// TIA Portal project "SWNC V1.0 pulldown" (V16)

(* hardware
DEVICE "S7-1200 station_1"  S7-1200 Station
   slot 0: "Rack_0"  S7-1200 Rack  Rack  V1.0
   slot 1: "PLC_1"  CPU 1214C DC/DC/DC  6ES7 214-1AG40-0XB0  V4.4
   slot 2: "DI 8x24VDC_1"  6ES7 221-1BF32-0XB0  V2.0
   slot 3: "CB 1241 (RS485)"  CB 1241 (RS485)  6ES7 241-1CH30-1XB0  V1.0
   slot 3: "DQ 8xRelay_1"  SM 1222 DQ8 x relay  6ES7 222-1HF32-0XB0  V2.0
   slot 4: "AI 8x13BIT_1"  6ES7 231-4HF32-0XB0  V2.1
   slot 5: "AQ 2x14BIT_1"  SM 1232 AQ2  6ES7 232-4HB32-0XB0  V2.1
DEVICE "HMI_1"  KTP700 Basic PN
   slot 0: "HMI_1"  KTP700 Basic PN  6AV2 123-2GB03-0AX0  16.0.0.0
   slot 1: "HMI_RT_1"  KTP700 Basic PN  6AV2 123-2GB03-0AX0  16.0.0.0
   slot 5: "HMI_1.IE_CP_1"  PROFINET Interface  16.0.0.0
      slot 1: "PROFINET Interface_1"  PROFINET Interface
         slot 1: "Port_1"  Port
*)

// ===== PLC "PLC_1"  CPU 1214C DC/DC/DC =====

VAR_GLOBAL   // PLC tag table "Default tag table"
   "HOA Manual" AT %I0.5 : Bool;
   "HOA Auto Run" AT %I0.4 : Bool;
   "supply empty" AT %I0.7 : Bool;
   "chiller full" AT %I1.0 : Bool;
   "chiller empty" AT %I1.1 : Bool;
   "inside full" AT %I1.3 : Bool;
   "inside discharge" AT %I1.4 : Bool;
   "inside empty" AT %I1.5 : Bool;
   "outside full" AT %I2.0 : Bool;
   "outside discharge" AT %I2.1 : Bool;
   "outside empty" AT %I2.2 : Bool;
   "purge full" AT %I1.2 : Bool;
   "E-Stop_Panel_pushed" AT %I0.6 : Bool;   // true when Estop is pushed
   "Run_button" AT %I0.0 : Bool;
   "Stop_reset_button" AT %I0.1 : Bool;
   "MAN 1 (Outside)" AT %Q0.0 : Bool;   // NO - to chiller NC - to purge
   "MAN 2 (Inside)" AT %Q0.1 : Bool;   // NO - to Purge NC - to Outside
   "MAN 3 (Supply)" AT %Q0.2 : Bool;   // NO - to outside NC - to inside
   "MAN 4 (Not Used)" AT %Q0.3 : Bool;   // NO - to outside NC - to inside
   "Pump 1 Outside cooling" AT %Q0.4 : Bool;
   "Pump 2 Outside Out" AT %Q0.5 : Bool;
   "Pump 3 Inside Cooling" AT %Q0.6 : Bool;
   "Pump 4 Inside Out" AT %Q0.7 : Bool;
   "Pump 5 Chiller out" AT %Q1.0 : Bool;
   "Pump 6 Supply out" AT %Q1.1 : Bool;
   "Pump 7 HX pump" AT %Q12.0 : Bool;
   "Pump 8 Purge out" AT %Q12.1 : Bool;
   "System_Byte" AT %MB1000 : Byte;
   "FirstScan" AT %M1000.0 : Bool;
   "DiagStatusUpdate" AT %M1000.1 : Bool;
   "AlwaysTRUE" AT %M1000.2 : Bool;
   "AlwaysFALSE" AT %M1000.3 : Bool;
   "Clock_Byte" AT %MB1001 : Byte;
   "Clock_10Hz" AT %M1001.0 : Bool;
   "Clock_5Hz" AT %M1001.1 : Bool;
   "Clock_2.5Hz" AT %M1001.2 : Bool;
   "Clock_2Hz" AT %M1001.3 : Bool;
   "Clock_1.25Hz" AT %M1001.4 : Bool;
   "Clock_1Hz" AT %M1001.5 : Bool;
   "Clock_0.625Hz" AT %M1001.6 : Bool;
   "Clock_0.5Hz" AT %M1001.7 : Bool;
   "Mode Bit" AT %MB0 : USInt;
   "HOA Off" AT %M1.0 : Bool;
   "Outside Fan" AT %M1.3 : Bool;
   "Inside Fan" AT %M1.4 : Bool;
   "Outside Cooling" AT %M1.5 : Bool;
   "Inside Cooling" AT %M1.6 : Bool;
   "pump out supply" AT %M1.7 : Bool;
   "pump out Chiller" AT %M2.0 : Bool;
   "pump out inside tank" AT %M2.1 : Bool;
   "Pump out outside tank" AT %M2.2 : Bool;
   "pump out purge tank" AT %M2.3 : Bool;
   "pump chiller circulation" AT %M2.4 : Bool;
   "valve from supply" AT %M2.5 : Bool;   // 0 = to outdoor 1= to indoor
   "valve from chiller" AT %M2.6 : Bool;   // 0 = to outdoor 1= to indoor
   "valve from inside" AT %M2.7 : Bool;   // 0 = to purge 1= to chiller
   "valve from outside" AT %M3.0 : Bool;   // 0 = to purge 1= to chiller
   "chiller enable" AT %M3.1 : Bool;
   "SB OUTSIDE COOLING" AT %M3.2 : Bool;
   "SB INSIDE COOLING" AT %M3.3 : Bool;
   "SB pump out supply" AT %M3.4 : Bool;
   "SB pump out Chiller" AT %M3.5 : Bool;
   "SB pump out inside tank" AT %M3.6 : Bool;
   "SB Pump out outside tank" AT %M3.7 : Bool;
   "SB pump out purge tank" AT %M4.0 : Bool;
   "SB pump chiller circulation" AT %M4.1 : Bool;
   "SB valve from supply" AT %M4.2 : Bool;
   "SB valve from chiller" AT %M4.3 : Bool;
   "SB valve from inside" AT %M4.4 : Bool;
   "SB valve from outside" AT %M4.5 : Bool;
   "SB chiller enable" AT %M4.6 : Bool;
   "SB INSIDE FAN" AT %M4.7 : Bool;
   "SB OUTSIDE FAN" AT %M5.0 : Bool;
   "inside change bit" AT %M5.1 : Bool;   // true when tank change is in progress
   "PB_chill to regen trans" AT %M5.2 : Bool;
   "PB_regen to chill trans" AT %M5.3 : Bool;
   "Emergency_flags" AT %MW6 : Int;   // Contain all the Estop scenarios. 1=active, 0=inactive
   "Emergency_check" AT %M7.0 : Bool;   // ON when any emergency scenario occurs
   "Emergency_Ack" AT %M1.2 : Bool;
   "Alarm_Ack" AT %MW1002 : Int;
   "global MB address" AT %MB8 : SInt;
   "GET_INT" AT %MW12 : Int;
   "HTS1" AT %M5.4 : Bool;   // Set bit for HT sensors
   "HTS3" AT %M5.6 : Bool;
   "HTS4" AT %M5.7 : Bool;
   "HTS2" AT %M9.0 : Bool;
   "DGS1" AT %M5.5 : Bool;   // Depth Gauge set bit
   "DGS2" AT %M9.1 : Bool;
   "WTSB" AT %M9.2 : Bool;   // Water temp set bit
   "THE TIME" AT %MD14 : Time_Of_Day;
   "Global GH Temp" AT %MD18 : Real;
   "Global GH Hum" AT %MD22 : Real;
   "Program Run" AT %M1.1 : Bool;
   "Regen bit" AT %M9.3 : Bool;
   "Auto time override" AT %M9.4 : Bool;
   "Manual day night toggle" AT %M9.5 : Bool;
   "Manual night to day trans" AT %M9.6 : Bool;
   "Manual day to night trans" AT %M9.7 : Bool;
   "time OS1" AT %M10.0 : Bool;
   "time OS2" AT %M10.1 : Bool;
   "time OS3" AT %M10.2 : Bool;
   "time OS4" AT %M10.3 : Bool;
   "WSSB" AT %M10.4 : Bool;
   "log start" AT %M10.5 : Bool;
   "log start lock" AT %M10.6 : Bool;
END_VAR

DATA_BLOCK "System Properties"   // DB1
{ S7_Optimized_Access := 'TRUE' }
VERSION : 0.1
   VAR
      "Time" : Struct
         "Current Time" : Time_Of_Day;
         "Night time start" : Time_Of_Day := TOD#20:00:00;
         "Night time end" : Time_Of_Day := TOD#06:00:00;
         "is it day???" : Bool;   // 1 = day, 0 = night
      END_STRUCT;
      "Situation Bits" : Struct
         HOA : Int;
         "Day Run" : Bool;
         "Night Run" : Bool;
         "Day Tank Change" : Int;
         "Night Regen Complete" : Bool;
         "Day/Night Transition Bit" : Int;   // 0= no trans 1= day to night 2= night to day
         "regen or chill" : Int;   // 0 = chill , 1 = regen 3 = transition in progress
         "chilling to regen transition" : Bool;
         "regen to chilling transition" : Bool;
      END_STRUCT;
      "Comment status" : String := 'Idle';
      "Comment DN" : String := 'Time Unknown';
   END_VAR
BEGIN
END_DATA_BLOCK

DATA_BLOCK "Outputs"   // DB2
{ S7_Optimized_Access := 'TRUE' }
VERSION : 0.1
   VAR
      Fans : Struct
         "Inside Fan" : Bool;
         "Outside Fan" : Bool;
      END_STRUCT;
      "Cooling Pad Pumps" : Struct
         "Inside Cooling" : Bool;
         "Outside Cooling" : Bool;
      END_STRUCT;
      Pumps : Struct
         "From Supply Tank" : Bool;
         "From Chiller Tank" : Bool;
         "From Inside Tank" : Bool;
         "From Outside Tank" : Bool;
         "From Purge Tank" : Bool;
         "Chiller Recirculation" : Bool;
      END_STRUCT;
      Valves : Struct
         "From Supply" : Bool;   // 0= to outdoor, 1= to indoor
         "From Chiller" : Bool;   // 0= to outdoor, 1= to indoor
         "From Indoor" : Bool;   // 0= to Purge, 1= to Chiller
         "From Outdoor" : Bool;   // 0= to Purge, 1= to Chiller
      END_STRUCT;
      Chiller : Struct
         "Chiller Enable" : Bool;
      END_STRUCT;
   END_VAR
BEGIN
END_DATA_BLOCK

DATA_BLOCK "Alarm Conditions"   // DB3
{ S7_Optimized_Access := 'TRUE' }
VERSION : 0.1
   VAR
      "E Stop Pushed" : Bool;
      "Pump Over run" : Bool;
      "Alarm bit" : Bool;
      "Alarm Reset" : Bool;
   END_VAR
BEGIN
END_DATA_BLOCK

DATA_BLOCK "What Time is it?_DB"   // DB4
{ S7_Optimized_Access := 'TRUE' }
VERSION : 0.1
// stored: InstanceOfName What Time is it?
"What Time is it?"
BEGIN
END_DATA_BLOCK

DATA_BLOCK "What mode_DB"   // DB5
{ S7_Optimized_Access := 'TRUE' }
VERSION : 0.1
// stored: InstanceOfName What mode
"What mode"
BEGIN
END_DATA_BLOCK

DATA_BLOCK "Manual Mode_DB"   // DB6
{ S7_Optimized_Access := 'TRUE' }
VERSION : 0.1
// stored: InstanceOfName Manual Mode
"Manual Mode"
BEGIN
END_DATA_BLOCK

DATA_BLOCK "Day Operation_DB"   // DB7
{ S7_Optimized_Access := 'TRUE' }
VERSION : 0.1
// stored: InstanceOfName Day Operation
"Day Operation"
BEGIN
END_DATA_BLOCK

DATA_BLOCK "Night Operation_DB"   // DB8
{ S7_Optimized_Access := 'TRUE' }
VERSION : 0.1
// stored: InstanceOfName Night Operation
"Night Operation"
BEGIN
END_DATA_BLOCK

DATA_BLOCK "Tank check_DB"   // DB9
{ S7_Optimized_Access := 'TRUE' }
VERSION : 0.1
// stored: InstanceOfName Tank check
"Tank check"
BEGIN
END_DATA_BLOCK

DATA_BLOCK "inside tank switch_DB"   // DB11
{ S7_Optimized_Access := 'TRUE' }
VERSION : 0.1
// stored: InstanceOfName inside tank switch
"inside tank switch"
BEGIN
END_DATA_BLOCK

DATA_BLOCK "Auto Run Program_DB"   // DB12
{ S7_Optimized_Access := 'TRUE' }
VERSION : 0.1
// stored: InstanceOfName Auto Run Program
"Auto Run Program"
BEGIN
END_DATA_BLOCK

DATA_BLOCK "Day to Night change_DB"   // DB13
{ S7_Optimized_Access := 'TRUE' }
VERSION : 0.1
// stored: InstanceOfName Day to Night change
"Day to Night change"
BEGIN
END_DATA_BLOCK

DATA_BLOCK "Night to Day change_DB"   // DB14
{ S7_Optimized_Access := 'TRUE' }
VERSION : 0.1
// stored: InstanceOfName Night to Day change
"Night to Day change"
BEGIN
END_DATA_BLOCK

DATA_BLOCK "Auto Time_DB"   // DB15
{ S7_Optimized_Access := 'TRUE' }
VERSION : 0.1
// stored: InstanceOfName Auto Time
"Auto Time"
BEGIN
END_DATA_BLOCK

DATA_BLOCK "Manual Time_DB"   // DB18
{ S7_Optimized_Access := 'TRUE' }
VERSION : 0.1
// stored: InstanceOfName Manual Time
"Manual Time"
BEGIN
END_DATA_BLOCK

DATA_BLOCK "Get Weather Station Data_DB"   // DB20
{ S7_Optimized_Access := 'TRUE' }
VERSION : 0.1
// stored: InstanceOfName Get Weather Station Data
"Get Weather Station Data"
BEGIN
END_DATA_BLOCK

DATA_BLOCK "Weather Station Data"   // DB21
{ S7_Optimized_Access := 'TRUE' }
VERSION : 0.1
   VAR
      "Air Temperature" : Real;
      "Air Humidity" : Real;
      "Air Pressure (mBar)" : Real;
      CO2 : Real;
      "PM 2.5" : Real;
      "PM 10" : Real;
      "PM 100" : Real;
      "Wind Speed" : Real;
      "Wind Direction" : Real;
      "Light Intensity (μmol/m^2.s)" : Real;
      "Current Rainfall" : Real;
   END_VAR
BEGIN
END_DATA_BLOCK

DATA_BLOCK "Emergency_Stop_DB"   // DB22
{ S7_Optimized_Access := 'TRUE' }
AUTHOR : FF
VERSION : 0.1
// stored: InstanceOfName Emergency_Stop
"Emergency_Stop"
BEGIN
END_DATA_BLOCK

DATA_BLOCK "MODBUS DATA"   // DB24
{ S7_Optimized_Access := 'FALSE' }
VERSION : 0.1
   VAR
      "Start up done" : Bool;
      "Master Busy" : Bool;
      "Master Done" : Bool;
      "Master Error" : Bool;
      "Slave Address" : Int;
      "Memory Address" : DInt;
      "read/write" : Int;
      "data length" : Int;
      "memory pointer" : Byte;
   END_VAR
BEGIN
END_DATA_BLOCK

DATA_BLOCK "Ts and Hs"   // DB26
{ S7_Optimized_Access := 'TRUE' }
VERSION : 0.1
   VAR
      "Ambient Temp" : Real;
      "Ambient Humidity" : Real;
      "GH Temp" : Real;
      "GH Humidity" : Real;
      "Outside Outlet Temp" : Real;
      "Outside Outlet  Humidity" : Real;
      "Inside Outlet Temp" : Real;
      "Inside Outlet Humidity" : Real;
      "Chiller Tank Water Temp" : Real;
   END_VAR
BEGIN
END_DATA_BLOCK

DATA_BLOCK "MODBUS REGISTER"   // DB27
{ S7_Optimized_Access := 'FALSE' }
VERSION : 0.1
   VAR
      "Incomiong/Outgoing data" : Array[0..20] of Int;
   END_VAR
BEGIN
END_DATA_BLOCK

DATA_BLOCK "MODBUS_DB"   // DB28
{ S7_Optimized_Access := 'TRUE' }
VERSION : 0.1
// stored: InstanceOfName MODBUS
"MODBUS"
BEGIN
END_DATA_BLOCK

DATA_BLOCK "Get Ts and Hs_DB"   // DB29
{ S7_Optimized_Access := 'TRUE' }
VERSION : 0.1
// stored: InstanceOfName Get Ts and Hs
"Get Ts and Hs"
BEGIN
END_DATA_BLOCK

DATA_BLOCK "Depth Readings"   // DB30
{ S7_Optimized_Access := 'TRUE' }
VERSION : 0.1
   VAR
      "Outside Tank Depth" : Real;
      "Inside Tank Depth" : Real;
   END_VAR
BEGIN
END_DATA_BLOCK

DATA_BLOCK "Get Depths_DB"   // DB32
{ S7_Optimized_Access := 'TRUE' }
VERSION : 0.1
// stored: InstanceOfName Get Depths
"Get Depths"
BEGIN
END_DATA_BLOCK

DATA_BLOCK "Get Water Temp_DB"   // DB33
{ S7_Optimized_Access := 'TRUE' }
VERSION : 0.1
// stored: InstanceOfName Get Water Temp
"Get Water Temp"
BEGIN
END_DATA_BLOCK

DATA_BLOCK "Setup"   // DB34
{ S7_Optimized_Access := 'TRUE' }
VERSION : 0.1
   VAR
      "Day Cooling on/off threshold" : Real := 20.0;
      "Night Cooling on/off threshold" : Real := 18.0;
      "Regen hum low" : Real := 35.0;
      "Regen hum high" : Real := 65.0;
      "Day Fan Speed" : Int := 6000;
      "Night Fan Speed" : Int := 1000;
   END_VAR
BEGIN
END_DATA_BLOCK

DATA_BLOCK "Update Outside Fan_DB"   // DB35
{ S7_Optimized_Access := 'TRUE' }
VERSION : 0.1
// stored: InstanceOfName Update Outside Fan
"Update Outside Fan"
BEGIN
END_DATA_BLOCK

DATA_BLOCK "Update Inside Fan_DB"   // DB36
{ S7_Optimized_Access := 'TRUE' }
VERSION : 0.1
// stored: InstanceOfName Update Inside Fan
"Update Inside Fan"
BEGIN
END_DATA_BLOCK

DATA_BLOCK "MODBUS_DB_1"   // DB37
{ S7_Optimized_Access := 'TRUE' }
VERSION : 0.1
// stored: InstanceOfName MODBUS
"MODBUS"
BEGIN
END_DATA_BLOCK

DATA_BLOCK "Inside Fan Emergancy_DB"   // DB38
{ S7_Optimized_Access := 'TRUE' }
VERSION : 0.1
// stored: InstanceOfName Inside Fan Emergancy
"Inside Fan Emergancy"
BEGIN
END_DATA_BLOCK

DATA_BLOCK "MODBUS_DB_2"   // DB39
{ S7_Optimized_Access := 'TRUE' }
VERSION : 0.1
// stored: InstanceOfName MODBUS
"MODBUS"
BEGIN
END_DATA_BLOCK

DATA_BLOCK "MODBUS_DB_3"   // DB40
{ S7_Optimized_Access := 'TRUE' }
VERSION : 0.1
// stored: InstanceOfName MODBUS
"MODBUS"
BEGIN
END_DATA_BLOCK

DATA_BLOCK "Outside Fan Emergancy_DB"   // DB41
{ S7_Optimized_Access := 'TRUE' }
VERSION : 0.1
// stored: InstanceOfName Outside Fan Emergancy
"Outside Fan Emergancy"
BEGIN
END_DATA_BLOCK

DATA_BLOCK "Update Outside Fan_DB_1"   // DB42
{ S7_Optimized_Access := 'TRUE' }
VERSION : 0.1
// stored: InstanceOfName Update Outside Fan
"Update Outside Fan"
BEGIN
END_DATA_BLOCK

DATA_BLOCK "MODBUS_DB_4"   // DB43
{ S7_Optimized_Access := 'TRUE' }
VERSION : 0.1
// stored: InstanceOfName MODBUS
"MODBUS"
BEGIN
END_DATA_BLOCK

DATA_BLOCK "Off Mode_DB"   // DB44
{ S7_Optimized_Access := 'TRUE' }
VERSION : 0.1
// stored: InstanceOfName Off Mode
"Off Mode"
BEGIN
END_DATA_BLOCK

DATA_BLOCK "Fan Speeds"   // DB48
{ S7_Optimized_Access := 'TRUE' }
VERSION : 0.1
   VAR
      "Inside Fan Speed" : Int := 6000;
      "Outside Fan Speed" : Int := 6000;
   END_VAR
BEGIN
END_DATA_BLOCK

DATA_BLOCK "Current States"   // DB49
{ S7_Optimized_Access := 'TRUE' }
VERSION : 0.1
BEGIN
END_DATA_BLOCK

DATA_BLOCK "From AWS"   // DB50
{ S7_Optimized_Access := 'TRUE' }
VERSION : 0.1
BEGIN
END_DATA_BLOCK

DATA_BLOCK "Data log setup"   // DB52
{ S7_Optimized_Access := 'TRUE' }
VERSION : 0.1
   VAR
      "name" : String := 'Ashs_Log_Overnight';
      ID : DInt;
      hedder : String := 'Out Temp,Out Hum,In Temp,In Hum';
      "data log data" : Struct
         data : Array[0..3] of Real;
      END_STRUCT;
      "start done" : Bool;
   END_VAR
BEGIN
END_DATA_BLOCK

DATA_BLOCK "Data logging main_DB"   // DB54
{ S7_Optimized_Access := 'TRUE' }
VERSION : 0.1
// stored: InstanceOfName Data logging main
"Data logging main"
BEGIN
END_DATA_BLOCK

// folder: System blocks/Program resources

DATA_BLOCK "IEC_Timer_0_DB"   // DB10
{ S7_Optimized_Access := 'TRUE' }
AUTHOR : Simatic
FAMILY : IEC
NAME : IEC_TMR
VERSION : 1.0
// stored: InstanceOfName IEC_TIMER
"IEC_TIMER"
BEGIN
END_DATA_BLOCK

DATA_BLOCK "IEC_Timer_0_DB_2"   // DB16
{ S7_Optimized_Access := 'TRUE' }
AUTHOR : Simatic
FAMILY : IEC
NAME : IEC_TMR
VERSION : 1.0
// stored: InstanceOfName IEC_TIMER
"IEC_TIMER"
BEGIN
END_DATA_BLOCK

DATA_BLOCK "IEC_Timer_0_DB_3"   // DB17
{ S7_Optimized_Access := 'TRUE' }
AUTHOR : Simatic
FAMILY : IEC
NAME : IEC_TMR
VERSION : 1.0
// stored: InstanceOfName IEC_TIMER
"IEC_TIMER"
BEGIN
END_DATA_BLOCK

DATA_BLOCK "IEC_Timer_0_DB_1"   // DB19
{ S7_Optimized_Access := 'TRUE' }
AUTHOR : Simatic
FAMILY : IEC
NAME : IEC_TMR
VERSION : 1.0
// stored: InstanceOfName IEC_TIMER
"IEC_TIMER"
BEGIN
END_DATA_BLOCK

DATA_BLOCK "IEC_Timer_0_DB_6"   // DB31
{ S7_Optimized_Access := 'TRUE' }
AUTHOR : Simatic
FAMILY : IEC
NAME : IEC_TMR
VERSION : 1.0
// stored: InstanceOfName IEC_TIMER
"IEC_TIMER"
BEGIN
END_DATA_BLOCK

DATA_BLOCK "IEC_Timer_0_DB_5"   // DB45
{ S7_Optimized_Access := 'TRUE' }
AUTHOR : Simatic
FAMILY : IEC
NAME : IEC_TMR
VERSION : 1.0
// stored: InstanceOfName IEC_TIMER
"IEC_TIMER"
BEGIN
END_DATA_BLOCK

DATA_BLOCK "IEC_Timer_0_DB_7"   // DB46
{ S7_Optimized_Access := 'TRUE' }
AUTHOR : Simatic
FAMILY : IEC
NAME : IEC_TMR
VERSION : 1.0
// stored: InstanceOfName IEC_TIMER
"IEC_TIMER"
BEGIN
END_DATA_BLOCK

DATA_BLOCK "IEC_Timer_0_DB_8"   // DB47
{ S7_Optimized_Access := 'TRUE' }
AUTHOR : Simatic
FAMILY : IEC
NAME : IEC_TMR
VERSION : 1.0
// stored: InstanceOfName IEC_TIMER
"IEC_TIMER"
BEGIN
END_DATA_BLOCK

// folder: (top level)

FUNCTION_BLOCK "What Time is it?"   // FB1, LAD
{ S7_Optimized_Access := 'TRUE' }
VERSION : 0.1
   VAR
      temp1 : DTL;
      OS1 : Bool;
      OS2 : Bool;
      LTNE : Bool;
      OS3 : Bool;
      OS4 : Bool;
      OS5 : Bool;
   END_VAR
   VAR_TEMP
      temp2 : Int;
   END_VAR
   VAR_TEMP   // added for the SCL form of the ladder/FBD networks
      _w1 : Bool;
   END_VAR
BEGIN

REGION Network 1
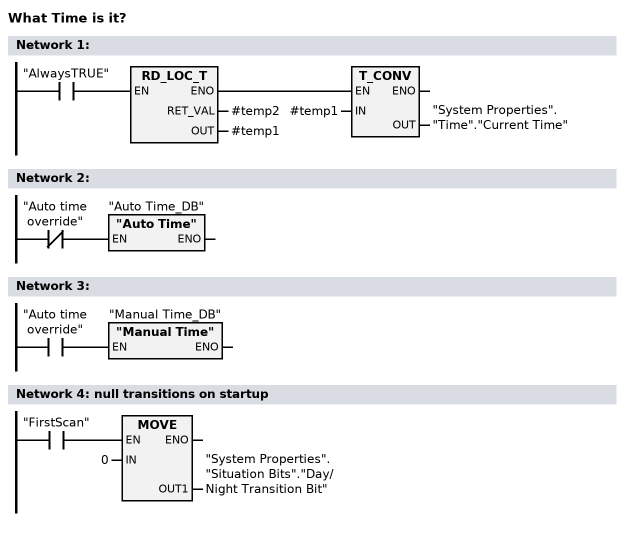
   // ENO of a box is taken as its EN; it also drops when the box reports an error
   #_w1 := "AlwaysTRUE";
   IF #_w1 THEN
       #temp2 := RD_LOC_T(OUT => #temp1);
       "System Properties"."Time"."Current Time" := T_CONV(IN := #temp1);
   END_IF;
END_REGION

REGION Network 2
   RUNG wire#powerrail
      I_Contact( "Auto time override" )
      "Auto Time_DB"()
   END_RUNG
   // the same network as SCL:
   IF NOT "Auto time override" THEN
       "Auto Time_DB"();   // "Auto Time"
   END_IF;
END_REGION

REGION Network 3
   RUNG wire#powerrail
      Contact( "Auto time override" )
      "Manual Time_DB"()
   END_RUNG
   // the same network as SCL:
   IF "Auto time override" THEN
       "Manual Time_DB"();   // "Manual Time"
   END_IF;
END_REGION

REGION Network 4: null transitions on startup
   RUNG wire#powerrail
      Contact( "FirstScan" )
      Move(in := 0, out1 => "System Properties"."Situation Bits"."Day/Night Transition Bit")
   END_RUNG
   // the same network as SCL:
   IF "FirstScan" THEN "System Properties"."Situation Bits"."Day/Night Transition Bit" := 0; END_IF;
END_REGION

REGION Network 5: 1 = day, 0 = night
END_REGION
END_FUNCTION_BLOCK

FUNCTION_BLOCK "What mode"   // FB2, LAD
{ S7_Optimized_Access := 'TRUE' }
VERSION : 0.1
   VAR_TEMP   // added for the SCL form of the ladder/FBD networks
      _w1 : Bool;
   END_VAR
BEGIN

REGION Network 1: Mode selection
   // 0 = startup
   // 1 = off
   // 2 = manual control
   // 3 = automatic run
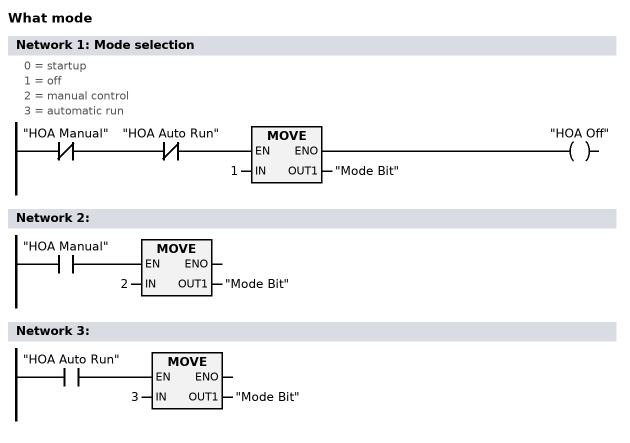
   RUNG wire#powerrail
      I_Contact( "HOA Manual" )
      I_Contact( "HOA Auto Run" )
      Move(in := 1, out1 => "Mode Bit")
      Coil( "HOA Off" )
   END_RUNG
   // the same network as SCL:
   #_w1 := NOT "HOA Manual" AND NOT "HOA Auto Run";
   IF #_w1 THEN "Mode Bit" := 1; END_IF;
   "HOA Off" := #_w1;
END_REGION

REGION Network 2
   RUNG wire#powerrail
      Contact( "HOA Manual" )
      Move(in := 2, out1 => "Mode Bit")
   END_RUNG
   // the same network as SCL:
   IF "HOA Manual" THEN "Mode Bit" := 2; END_IF;
END_REGION

REGION Network 3
   RUNG wire#powerrail
      Contact( "HOA Auto Run" )
      Move(in := 3, out1 => "Mode Bit")
   END_RUNG
   // the same network as SCL:
   IF "HOA Auto Run" THEN "Mode Bit" := 3; END_IF;
END_REGION
END_FUNCTION_BLOCK

FUNCTION_BLOCK "Manual Mode"   // FB3, LAD
{ S7_Optimized_Access := 'TRUE' }
VERSION : 0.1
BEGIN

REGION Network 1: Manual operation of outputs
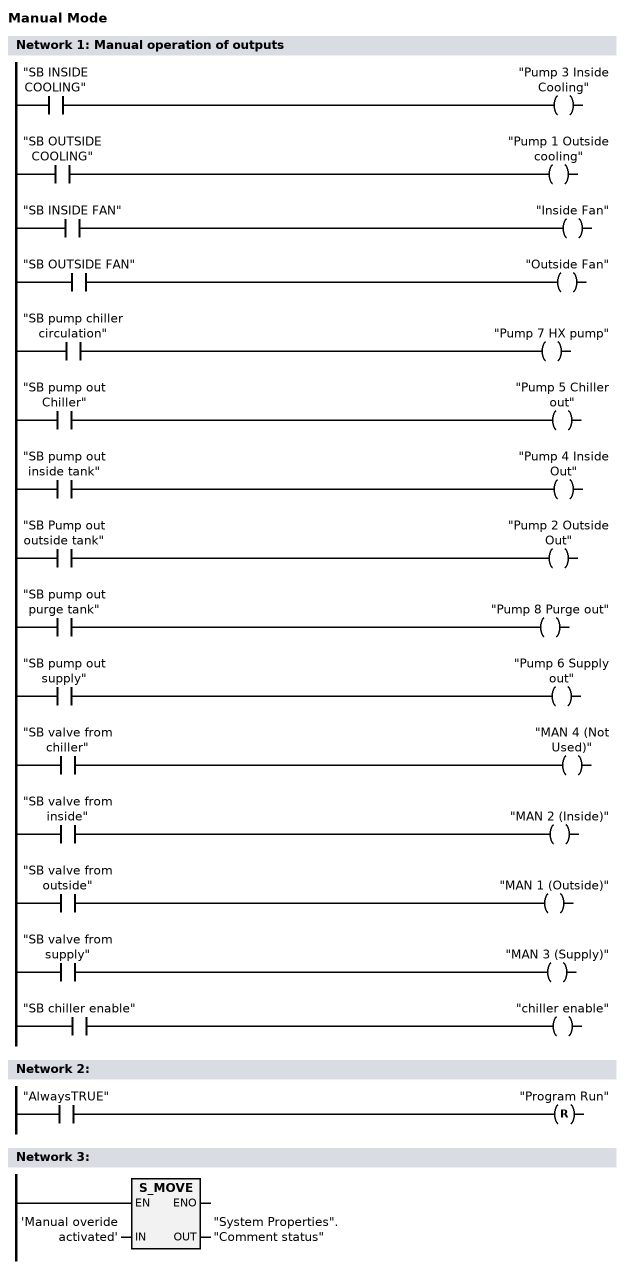
   RUNG wire#powerrail
      Contact( "SB INSIDE COOLING" )
      Coil( "Pump 3 Inside Cooling" )
   END_RUNG
   RUNG wire#powerrail
      Contact( "SB OUTSIDE COOLING" )
      Coil( "Pump 1 Outside cooling" )
   END_RUNG
   RUNG wire#powerrail
      Contact( "SB INSIDE FAN" )
      Coil( "Inside Fan" )
   END_RUNG
   RUNG wire#powerrail
      Contact( "SB OUTSIDE FAN" )
      Coil( "Outside Fan" )
   END_RUNG
   RUNG wire#powerrail
      Contact( "SB pump chiller circulation" )
      Coil( "Pump 7 HX pump" )
   END_RUNG
   RUNG wire#powerrail
      Contact( "SB pump out Chiller" )
      Coil( "Pump 5 Chiller out" )
   END_RUNG
   RUNG wire#powerrail
      Contact( "SB pump out inside tank" )
      Coil( "Pump 4 Inside Out" )
   END_RUNG
   RUNG wire#powerrail
      Contact( "SB Pump out outside tank" )
      Coil( "Pump 2 Outside Out" )
   END_RUNG
   RUNG wire#powerrail
      Contact( "SB pump out purge tank" )
      Coil( "Pump 8 Purge out" )
   END_RUNG
   RUNG wire#powerrail
      Contact( "SB pump out supply" )
      Coil( "Pump 6 Supply out" )
   END_RUNG
   RUNG wire#powerrail
      Contact( "SB valve from chiller" )
      Coil( "MAN 4 (Not Used)" )
   END_RUNG
   RUNG wire#powerrail
      Contact( "SB valve from inside" )
      Coil( "MAN 2 (Inside)" )
   END_RUNG
   RUNG wire#powerrail
      Contact( "SB valve from outside" )
      Coil( "MAN 1 (Outside)" )
   END_RUNG
   RUNG wire#powerrail
      Contact( "SB valve from supply" )
      Coil( "MAN 3 (Supply)" )
   END_RUNG
   RUNG wire#powerrail
      Contact( "SB chiller enable" )
      Coil( "chiller enable" )
   END_RUNG
   // the same network as SCL:
   "Pump 3 Inside Cooling" := "SB INSIDE COOLING";
   "Pump 1 Outside cooling" := "SB OUTSIDE COOLING";
   "Inside Fan" := "SB INSIDE FAN";
   "Outside Fan" := "SB OUTSIDE FAN";
   "Pump 7 HX pump" := "SB pump chiller circulation";
   "Pump 5 Chiller out" := "SB pump out Chiller";
   "Pump 4 Inside Out" := "SB pump out inside tank";
   "Pump 2 Outside Out" := "SB Pump out outside tank";
   "Pump 8 Purge out" := "SB pump out purge tank";
   "Pump 6 Supply out" := "SB pump out supply";
   "MAN 4 (Not Used)" := "SB valve from chiller";
   "MAN 2 (Inside)" := "SB valve from inside";
   "MAN 1 (Outside)" := "SB valve from outside";
   "MAN 3 (Supply)" := "SB valve from supply";
   "chiller enable" := "SB chiller enable";
END_REGION

REGION Network 2
   RUNG wire#powerrail
      Contact( "AlwaysTRUE" )
      R_Coil( "Program Run" )
   END_RUNG
   // the same network as SCL:
   IF "AlwaysTRUE" THEN "Program Run" := FALSE; END_IF;
END_REGION

REGION Network 3
   RUNG wire#powerrail
      S_Move(in := 'Manual overide activated', out => "System Properties"."Comment status")
   END_RUNG
   // the same network as SCL:
   "System Properties"."Comment status" := 'Manual overide activated';
END_REGION
END_FUNCTION_BLOCK

FUNCTION_BLOCK "Auto Run Program"   // FB4, LAD
{ S7_Optimized_Access := 'TRUE' }
VERSION : 0.1
BEGIN

REGION Network 1: Select for day or night operation
   // only works when there is not transitions happening
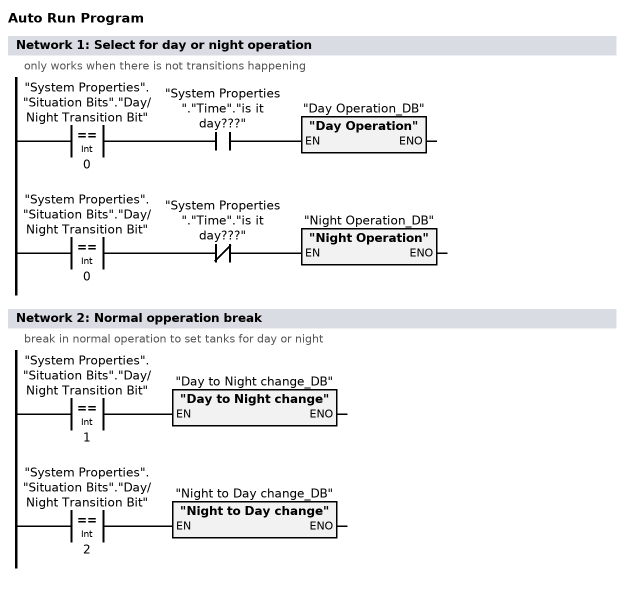
   RUNG wire#powerrail
      { S7_Templates := "SrcType := Int" } EQ_Contact(in1 := "System Properties"."Situation Bits"."Day/Night Transition Bit", in2 := 0)
      Contact( "System Properties"."Time"."is it day???" )
      "Day Operation_DB"()
   END_RUNG
   RUNG wire#powerrail
      { S7_Templates := "SrcType := Int" } EQ_Contact(in1 := "System Properties"."Situation Bits"."Day/Night Transition Bit", in2 := 0)
      I_Contact( "System Properties"."Time"."is it day???" )
      "Night Operation_DB"()
   END_RUNG
   // the same network as SCL:
   IF ("System Properties"."Situation Bits"."Day/Night Transition Bit" = 0) AND "System Properties"."Time"."is it day???" THEN
       "Day Operation_DB"();   // "Day Operation"
   END_IF;
   IF ("System Properties"."Situation Bits"."Day/Night Transition Bit" = 0) AND NOT "System Properties"."Time"."is it day???" THEN
       "Night Operation_DB"();   // "Night Operation"
   END_IF;
END_REGION

REGION Network 2: Normal opperation break
   // break in normal operation to set tanks for day or night
   RUNG wire#powerrail
      { S7_Templates := "SrcType := Int" } EQ_Contact(in1 := "System Properties"."Situation Bits"."Day/Night Transition Bit", in2 := 1)
      "Day to Night change_DB"()
   END_RUNG
   RUNG wire#powerrail
      { S7_Templates := "SrcType := Int" } EQ_Contact(in1 := "System Properties"."Situation Bits"."Day/Night Transition Bit", in2 := 2)
      "Night to Day change_DB"()
   END_RUNG
   // the same network as SCL:
   IF "System Properties"."Situation Bits"."Day/Night Transition Bit" = 1 THEN
       "Day to Night change_DB"();   // "Day to Night change"
   END_IF;
   IF "System Properties"."Situation Bits"."Day/Night Transition Bit" = 2 THEN
       "Night to Day change_DB"();   // "Night to Day change"
   END_IF;
END_REGION
END_FUNCTION_BLOCK

FUNCTION_BLOCK "Day Operation"   // FB5, LAD
{ S7_Optimized_Access := 'TRUE' }
VERSION : 0.1
BEGIN

REGION Network 1: SW cooling if GH temp is above setpoint and speed set
   // to make VFD control
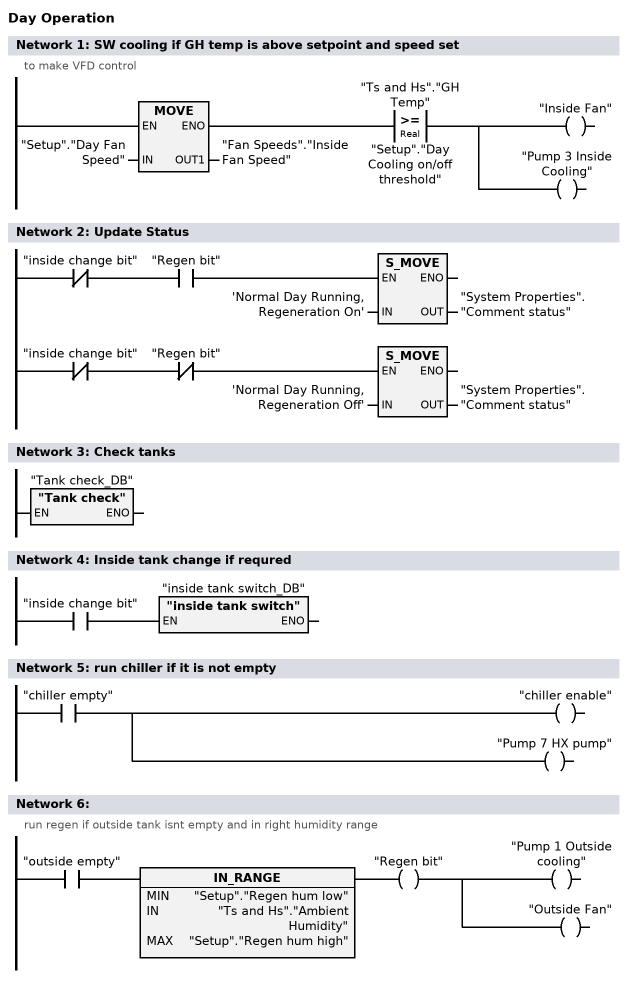
   RUNG wire#powerrail
      Move(in := "Setup"."Day Fan Speed", out1 => "Fan Speeds"."Inside Fan Speed")
      { S7_Templates := "SrcType := Real" } GE_Contact(in1 := "Ts and Hs"."GH Temp", in2 := "Setup"."Day Cooling on/off threshold")
      wire#w1
      Coil( "Inside Fan" )
   END_RUNG
   RUNG wire#w1
      Coil( "Pump 3 Inside Cooling" )
   END_RUNG
   // the same network as SCL:
   "Fan Speeds"."Inside Fan Speed" := "Setup"."Day Fan Speed";
   "Inside Fan" := "Ts and Hs"."GH Temp" >= "Setup"."Day Cooling on/off threshold";
   "Pump 3 Inside Cooling" := "Inside Fan";
END_REGION

REGION Network 2: Update Status
   RUNG wire#powerrail
      I_Contact( "inside change bit" )
      Contact( "Regen bit" )
      S_Move(in := 'Normal Day Running, Regeneration On', out => "System Properties"."Comment status")
   END_RUNG
   RUNG wire#powerrail
      I_Contact( "inside change bit" )
      I_Contact( "Regen bit" )
      S_Move(in := 'Normal Day Running, Regeneration Off', out => "System Properties"."Comment status")
   END_RUNG
   // the same network as SCL:
   IF NOT "inside change bit" AND "Regen bit" THEN
       "System Properties"."Comment status" := 'Normal Day Running, Regeneration On';
   END_IF;
   IF NOT "inside change bit" AND NOT "Regen bit" THEN
       "System Properties"."Comment status" := 'Normal Day Running, Regeneration Off';
   END_IF;
END_REGION

REGION Network 3: Check tanks
   RUNG wire#powerrail
      "Tank check_DB"()
   END_RUNG
   // the same network as SCL:
   "Tank check_DB"();   // "Tank check"
END_REGION

REGION Network 4: Inside tank change if requred
   RUNG wire#powerrail
      Contact( "inside change bit" )
      "inside tank switch_DB"()
   END_RUNG
   // the same network as SCL:
   IF "inside change bit" THEN
       "inside tank switch_DB"();   // "inside tank switch"
   END_IF;
END_REGION

REGION Network 5: run chiller if it is not empty
   RUNG wire#powerrail
      Contact( "chiller empty" )
      wire#w1
      Coil( "chiller enable" )
   END_RUNG
   RUNG wire#w1
      Coil( "Pump 7 HX pump" )
   END_RUNG
   // the same network as SCL:
   "chiller enable" := "chiller empty";
   "Pump 7 HX pump" := "chiller empty";
END_REGION

REGION Network 6
   // run regen if outside tank isnt empty and in right humidity range
   RUNG wire#powerrail
      Contact( "outside empty" )
      { S7_Templates := "SrcType := Real" } InRange(min := "Setup"."Regen hum low", in := "Ts and Hs"."Ambient Humidity", max := "Setup"."Regen hum high")
      Coil( "Regen bit" )
      wire#w1
      Coil( "Pump 1 Outside cooling" )
   END_RUNG
   RUNG wire#w1
      Coil( "Outside Fan" )
   END_RUNG
   // the same network as SCL:
   "Regen bit" := "outside empty" AND ("Setup"."Regen hum low" <= "Ts and Hs"."Ambient Humidity") AND ("Ts and Hs"."Ambient Humidity" <= "Setup"."Regen hum high");
   "Pump 1 Outside cooling" := "Regen bit";
   "Outside Fan" := "Regen bit";
END_REGION

REGION Network 7: set regen or chill to 3 and select mode to force transition (to be done in HMI)
END_REGION
END_FUNCTION_BLOCK

FUNCTION_BLOCK "Night Operation"   // FB6, LAD
{ S7_Optimized_Access := 'TRUE' }
VERSION : 0.1
BEGIN

REGION Network 1
   // Run night chilling if inside not empty and is above temp setpoint and speed set
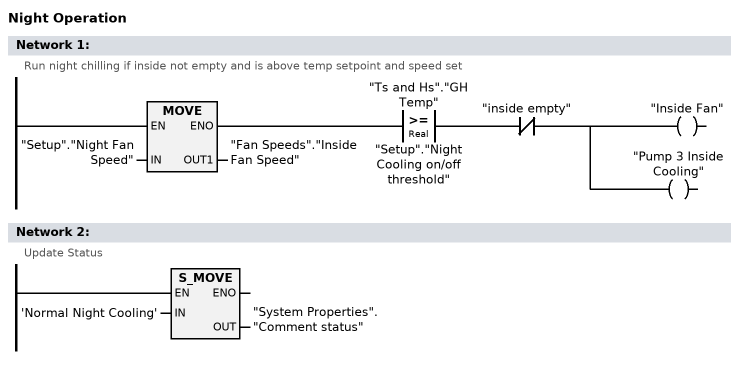
   RUNG wire#powerrail
      Move(in := "Setup"."Night Fan Speed", out1 => "Fan Speeds"."Inside Fan Speed")
      { S7_Templates := "SrcType := Real" } GE_Contact(in1 := "Ts and Hs"."GH Temp", in2 := "Setup"."Night Cooling on/off threshold")
      I_Contact( "inside empty" )
      wire#w1
      Coil( "Inside Fan" )
   END_RUNG
   RUNG wire#w1
      Coil( "Pump 3 Inside Cooling" )
   END_RUNG
   // the same network as SCL:
   "Fan Speeds"."Inside Fan Speed" := "Setup"."Night Fan Speed";
   "Inside Fan" := ("Ts and Hs"."GH Temp" >= "Setup"."Night Cooling on/off threshold") AND NOT "inside empty";
   "Pump 3 Inside Cooling" := "Inside Fan";
END_REGION

REGION Network 2
   // Update Status
   RUNG wire#powerrail
      S_Move(in := 'Normal Night Cooling', out => "System Properties"."Comment status")
   END_RUNG
   // the same network as SCL:
   "System Properties"."Comment status" := 'Normal Night Cooling';
END_REGION
END_FUNCTION_BLOCK

FUNCTION_BLOCK "Tank check"   // FB7, LAD
{ S7_Optimized_Access := 'TRUE' }
VERSION : 0.1
BEGIN

REGION Network 1: sets to true when the inside tank hits its discharge level
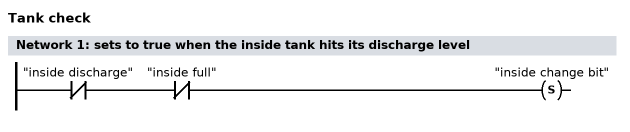
   RUNG wire#powerrail
      I_Contact( "inside discharge" )
      I_Contact( "inside full" )
      S_Coil( "inside change bit" )
   END_RUNG
   // the same network as SCL:
   IF NOT "inside discharge" AND NOT "inside full" THEN "inside change bit" := TRUE; END_IF;
END_REGION
END_FUNCTION_BLOCK

FUNCTION_BLOCK "inside tank switch"   // FB8, LAD
{ S7_Optimized_Access := 'TRUE' }
VERSION : 0.1
   VAR_TEMP   // added for the SCL form of the ladder/FBD networks
      _w1 : Bool;
   END_VAR
BEGIN

REGION Network 1: valve set up --- 0 = to outside 1= to purge
   // set to purge (valve is not energised)
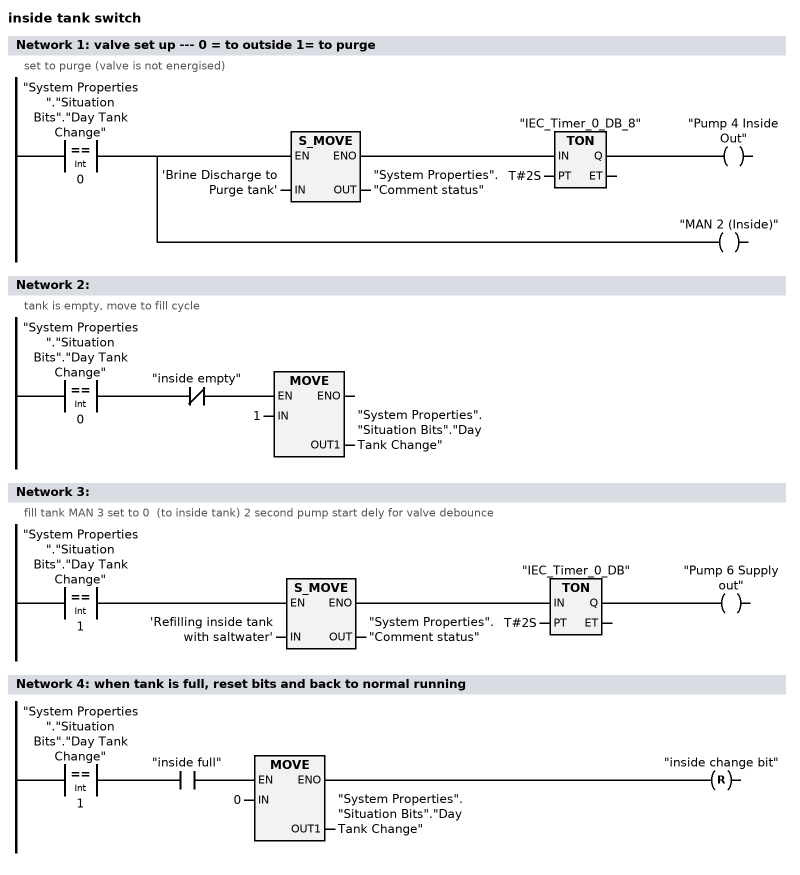
   #_w1 := "System Properties"."Situation Bits"."Day Tank Change" = 0;
   IF #_w1 THEN "System Properties"."Comment status" := 'Brine Discharge to Purge tank'; END_IF;
   "IEC_Timer_0_DB_8".TON(IN := #_w1, PT := T#2S);
   "Pump 4 Inside Out" := "IEC_Timer_0_DB_8".Q;
   "MAN 2 (Inside)" := #_w1;
END_REGION

REGION Network 2
   // tank is empty, move to fill cycle
   RUNG wire#powerrail
      { S7_Templates := "SrcType := Int" } EQ_Contact(in1 := "System Properties"."Situation Bits"."Day Tank Change", in2 := 0)
      I_Contact( "inside empty" )
      Move(in := 1, out1 => "System Properties"."Situation Bits"."Day Tank Change")
   END_RUNG
   // the same network as SCL:
   IF ("System Properties"."Situation Bits"."Day Tank Change" = 0) AND NOT "inside empty" THEN
       "System Properties"."Situation Bits"."Day Tank Change" := 1;
   END_IF;
END_REGION

REGION Network 3
   // fill tank MAN 3 set to 0  (to inside tank) 2 second pump start dely for valve debounce
   #_w1 := "System Properties"."Situation Bits"."Day Tank Change" = 1;
   IF #_w1 THEN "System Properties"."Comment status" := 'Refilling inside tank with saltwater'; END_IF;
   "IEC_Timer_0_DB".TON(IN := #_w1, PT := T#2S);
   "Pump 6 Supply out" := "IEC_Timer_0_DB".Q;
END_REGION

REGION Network 4: when tank is full, reset bits and back to normal running
   RUNG wire#powerrail
      { S7_Templates := "SrcType := Int" } EQ_Contact(in1 := "System Properties"."Situation Bits"."Day Tank Change", in2 := 1)
      Contact( "inside full" )
      Move(in := 0, out1 => "System Properties"."Situation Bits"."Day Tank Change")
      R_Coil( "inside change bit" )
   END_RUNG
   // the same network as SCL:
   #_w1 := ("System Properties"."Situation Bits"."Day Tank Change" = 1) AND "inside full";
   IF #_w1 THEN
       "System Properties"."Situation Bits"."Day Tank Change" := 0;
       "inside change bit" := FALSE;
   END_IF;
END_REGION
END_FUNCTION_BLOCK

FUNCTION_BLOCK "Day to Night change"   // FB9, LAD
{ S7_Optimized_Access := 'TRUE' }
VERSION : 0.1
   VAR
      "DN change bit" : Int;
   END_VAR
   VAR_TEMP   // added for the SCL form of the ladder/FBD networks
      _w1 : Bool;
   END_VAR
BEGIN

REGION Network 1
   // inside tank to purge (valve at 1) 2 second debounce
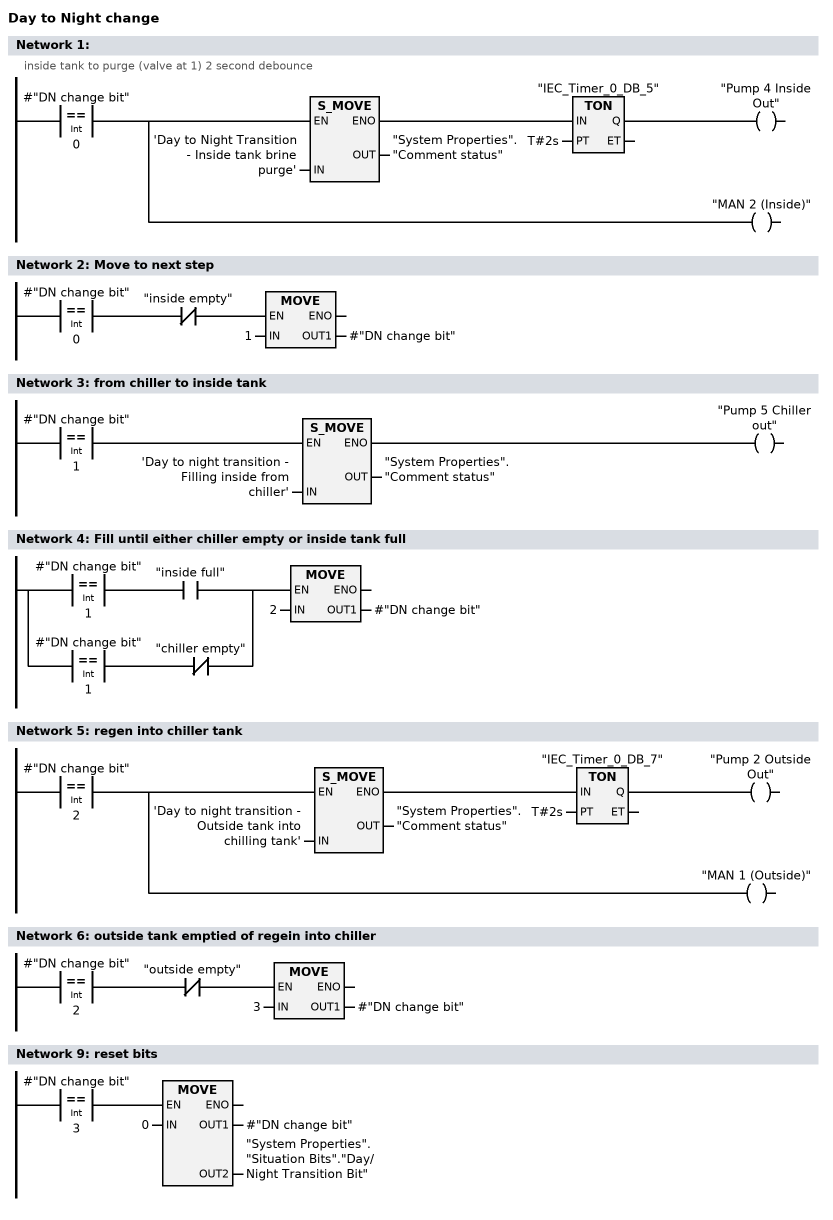
   #_w1 := #"DN change bit" = 0;
   IF #_w1 THEN
       "System Properties"."Comment status" := 'Day to Night Transition - Inside tank brine purge';
   END_IF;
   "IEC_Timer_0_DB_5".TON(IN := #_w1, PT := T#2s);
   "Pump 4 Inside Out" := "IEC_Timer_0_DB_5".Q;
   "MAN 2 (Inside)" := #_w1;
END_REGION

REGION Network 2: Move to next step
   RUNG wire#powerrail
      { S7_Templates := "SrcType := Int" } EQ_Contact(in1 := #"DN change bit", in2 := 0)
      I_Contact( "inside empty" )
      Move(in := 1, out1 => #"DN change bit")
   END_RUNG
   // the same network as SCL:
   IF (#"DN change bit" = 0) AND NOT "inside empty" THEN #"DN change bit" := 1; END_IF;
END_REGION

REGION Network 3: from chiller to inside tank
   RUNG wire#powerrail
      { S7_Templates := "SrcType := Int" } EQ_Contact(in1 := #"DN change bit", in2 := 1)
      S_Move(in := 'Day to night transition - Filling inside from chiller', out => "System Properties"."Comment status")
      Coil( "Pump 5 Chiller out" )
   END_RUNG
   // the same network as SCL:
   #_w1 := #"DN change bit" = 1;
   IF #_w1 THEN
       "System Properties"."Comment status" := 'Day to night transition - Filling inside from chiller';
   END_IF;
   "Pump 5 Chiller out" := #_w1;
END_REGION

REGION Network 4: Fill until either chiller empty or inside tank full
   RUNG wire#powerrail
      { S7_Templates := "SrcType := Int" } EQ_Contact(in1 := #"DN change bit", in2 := 1)
      Contact( "inside full" )
      wire#w1
      Move(in := 2, out1 => #"DN change bit")
   END_RUNG
   RUNG wire#powerrail
      { S7_Templates := "SrcType := Int" } EQ_Contact(in1 := #"DN change bit", in2 := 1)
      I_Contact( "chiller empty" )
   END_RUNG wire#w1
   // the same network as SCL:
   IF ((#"DN change bit" = 1) AND "inside full") OR ((#"DN change bit" = 1) AND NOT "chiller empty") THEN
       #"DN change bit" := 2;
   END_IF;
END_REGION

REGION Network 5: regen into chiller tank
   #_w1 := #"DN change bit" = 2;
   IF #_w1 THEN
       "System Properties"."Comment status" := 'Day to night transition - Outside tank into chilling tank';
   END_IF;
   "IEC_Timer_0_DB_7".TON(IN := #_w1, PT := T#2s);
   "Pump 2 Outside Out" := "IEC_Timer_0_DB_7".Q;
   "MAN 1 (Outside)" := #_w1;
END_REGION

REGION Network 6: outside tank emptied of regein into chiller
   RUNG wire#powerrail
      { S7_Templates := "SrcType := Int" } EQ_Contact(in1 := #"DN change bit", in2 := 2)
      I_Contact( "outside empty" )
      Move(in := 3, out1 => #"DN change bit")
   END_RUNG
   // the same network as SCL:
   IF (#"DN change bit" = 2) AND NOT "outside empty" THEN #"DN change bit" := 3; END_IF;
END_REGION

REGION Network 9: reset bits
   RUNG wire#powerrail
      { S7_Templates := "SrcType := Int" } EQ_Contact(in1 := #"DN change bit", in2 := 3)
      Move(in := 0, out1 => #"DN change bit", out2 => "System Properties"."Situation Bits"."Day/Night Transition Bit")
   END_RUNG
   // the same network as SCL:
   IF #"DN change bit" = 3 THEN
       #"DN change bit" := 0;
       "System Properties"."Situation Bits"."Day/Night Transition Bit" := 0;
   END_IF;
END_REGION
END_FUNCTION_BLOCK

FUNCTION_BLOCK "Night to Day change"   // FB10, LAD
{ S7_Optimized_Access := 'TRUE' }
VERSION : 0.1
   VAR
      "ND change bit" : Int;
   END_VAR
   VAR_TEMP   // added for the SCL form of the ladder/FBD networks
      _w1 : Bool;
   END_VAR
BEGIN

REGION Network 1: move from inside back to outside, MAN 2 at 0 (to outside)
   // 2 second valve debounce
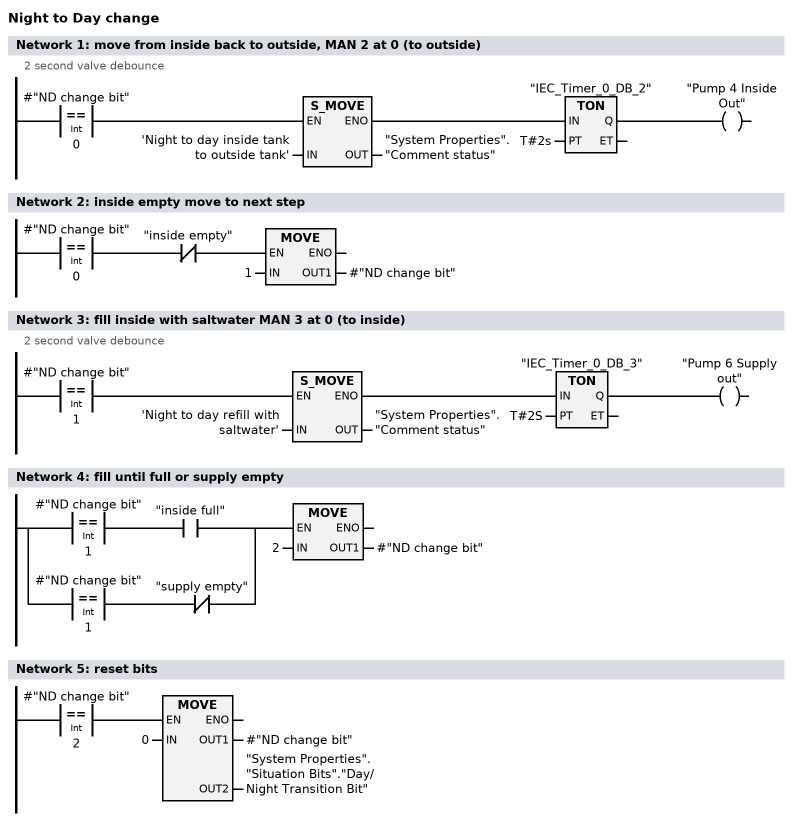
   #_w1 := #"ND change bit" = 0;
   IF #_w1 THEN "System Properties"."Comment status" := 'Night to day inside tank to outside tank'; END_IF;
   "IEC_Timer_0_DB_2".TON(IN := #_w1, PT := T#2s);
   "Pump 4 Inside Out" := "IEC_Timer_0_DB_2".Q;
END_REGION

REGION Network 2: inside empty move to next step
   RUNG wire#powerrail
      { S7_Templates := "SrcType := Int" } EQ_Contact(in1 := #"ND change bit", in2 := 0)
      I_Contact( "inside empty" )
      Move(in := 1, out1 => #"ND change bit")
   END_RUNG
   // the same network as SCL:
   IF (#"ND change bit" = 0) AND NOT "inside empty" THEN #"ND change bit" := 1; END_IF;
END_REGION

REGION Network 3: fill inside with saltwater MAN 3 at 0 (to inside)
   // 2 second valve debounce
   #_w1 := #"ND change bit" = 1;
   IF #_w1 THEN "System Properties"."Comment status" := 'Night to day refill with saltwater'; END_IF;
   "IEC_Timer_0_DB_3".TON(IN := #_w1, PT := T#2S);
   "Pump 6 Supply out" := "IEC_Timer_0_DB_3".Q;
END_REGION

REGION Network 4: fill until full or supply empty
   RUNG wire#powerrail
      { S7_Templates := "SrcType := Int" } EQ_Contact(in1 := #"ND change bit", in2 := 1)
      Contact( "inside full" )
      wire#w1
      Move(in := 2, out1 => #"ND change bit")
   END_RUNG
   RUNG wire#powerrail
      { S7_Templates := "SrcType := Int" } EQ_Contact(in1 := #"ND change bit", in2 := 1)
      I_Contact( "supply empty" )
   END_RUNG wire#w1
   // the same network as SCL:
   IF ((#"ND change bit" = 1) AND "inside full") OR ((#"ND change bit" = 1) AND NOT "supply empty") THEN
       #"ND change bit" := 2;
   END_IF;
END_REGION

REGION Network 5: reset bits
   RUNG wire#powerrail
      { S7_Templates := "SrcType := Int" } EQ_Contact(in1 := #"ND change bit", in2 := 2)
      Move(in := 0, out1 => #"ND change bit", out2 => "System Properties"."Situation Bits"."Day/Night Transition Bit")
   END_RUNG
   // the same network as SCL:
   IF #"ND change bit" = 2 THEN
       #"ND change bit" := 0;
       "System Properties"."Situation Bits"."Day/Night Transition Bit" := 0;
   END_IF;
END_REGION
END_FUNCTION_BLOCK

FUNCTION_BLOCK "Auto Time"   // FB11, LAD
{ S7_Optimized_Access := 'TRUE' }
VERSION : 0.1
   VAR_TEMP   // added for the SCL form of the ladder/FBD networks
      _w1 : Bool;
      _w2 : Bool;
      _w3 : Bool;
      _w4 : Bool;
   END_VAR
BEGIN

REGION Network 2: 1 = day, 0 = night
   // also set the day/night transition integer
   // 0 = no transition
   // 1 = day to night transition
   // 2 = night to day transition
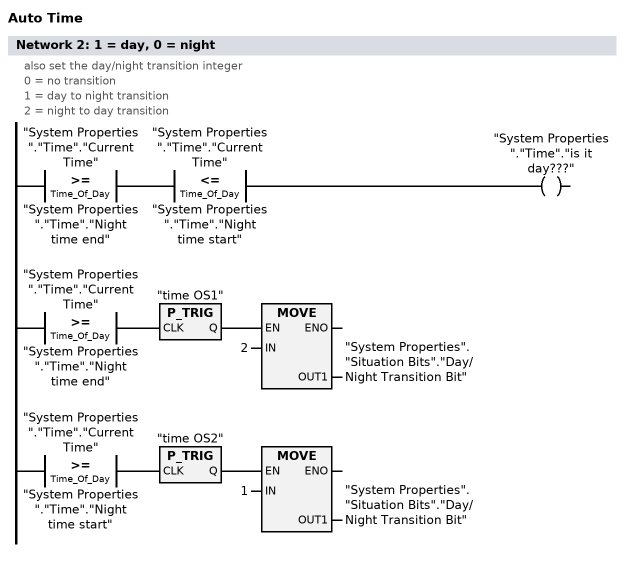
   RUNG wire#powerrail
      { S7_Templates := "SrcType := Time_Of_Day" } GE_Contact(in1 := "System Properties"."Time"."Current Time", in2 := "System Properties"."Time"."Night time end")
      { S7_Templates := "SrcType := Time_Of_Day" } LE_Contact(in1 := "System Properties"."Time"."Current Time", in2 := "System Properties"."Time"."Night time start")
      Coil( "System Properties"."Time"."is it day???" )
   END_RUNG
   RUNG wire#powerrail
      { S7_Templates := "SrcType := Time_Of_Day" } GE_Contact(in1 := "System Properties"."Time"."Current Time", in2 := "System Properties"."Time"."Night time end")
      P_Trig( "time OS1" )
      Move(in := 2, out1 => "System Properties"."Situation Bits"."Day/Night Transition Bit")
   END_RUNG
   RUNG wire#powerrail
      { S7_Templates := "SrcType := Time_Of_Day" } GE_Contact(in1 := "System Properties"."Time"."Current Time", in2 := "System Properties"."Time"."Night time start")
      P_Trig( "time OS2" )
      Move(in := 1, out1 => "System Properties"."Situation Bits"."Day/Night Transition Bit")
   END_RUNG
   // the same network as SCL:
   "System Properties"."Time"."is it day???" := ("System Properties"."Time"."Current Time" >= "System Properties"."Time"."Night time end") AND ("System Properties"."Time"."Current Time" <= "System Properties"."Time"."Night time start");
   #_w1 := "System Properties"."Time"."Current Time" >= "System Properties"."Time"."Night time end";
   #_w2 := #_w1 AND NOT "time OS1";   // rising edge
   "time OS1" := #_w1;
   IF #_w2 THEN "System Properties"."Situation Bits"."Day/Night Transition Bit" := 2; END_IF;
   #_w3 := "System Properties"."Time"."Current Time" >= "System Properties"."Time"."Night time start";
   #_w4 := #_w3 AND NOT "time OS2";   // rising edge
   "time OS2" := #_w3;
   IF #_w4 THEN "System Properties"."Situation Bits"."Day/Night Transition Bit" := 1; END_IF;
END_REGION
END_FUNCTION_BLOCK

FUNCTION_BLOCK "Manual Time"   // FB12, LAD
{ S7_Optimized_Access := 'TRUE' }
VERSION : 0.1
   VAR_TEMP   // added for the SCL form of the ladder/FBD networks
      _w1 : Bool;
      _w2 : Bool;
   END_VAR
BEGIN

REGION Network 1: 1 = day, 0 = night
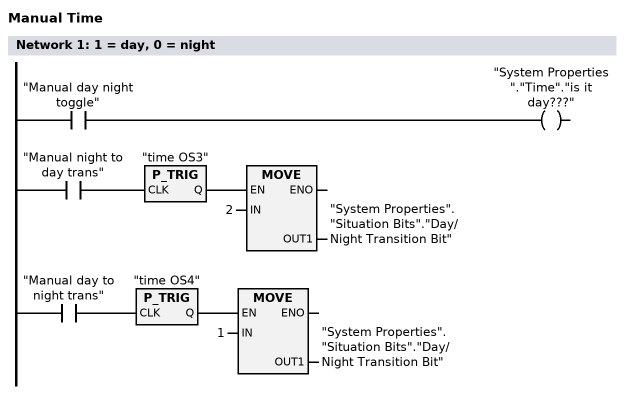
   RUNG wire#powerrail
      Contact( "Manual day night toggle" )
      Coil( "System Properties"."Time"."is it day???" )
   END_RUNG
   RUNG wire#powerrail
      Contact( "Manual night to day trans" )
      P_Trig( "time OS3" )
      Move(in := 2, out1 => "System Properties"."Situation Bits"."Day/Night Transition Bit")
   END_RUNG
   RUNG wire#powerrail
      Contact( "Manual day to night trans" )
      P_Trig( "time OS4" )
      Move(in := 1, out1 => "System Properties"."Situation Bits"."Day/Night Transition Bit")
   END_RUNG
   // the same network as SCL:
   "System Properties"."Time"."is it day???" := "Manual day night toggle";
   #_w1 := "Manual night to day trans" AND NOT "time OS3";   // rising edge
   "time OS3" := "Manual night to day trans";
   IF #_w1 THEN "System Properties"."Situation Bits"."Day/Night Transition Bit" := 2; END_IF;
   #_w2 := "Manual day to night trans" AND NOT "time OS4";   // rising edge
   "time OS4" := "Manual day to night trans";
   IF #_w2 THEN "System Properties"."Situation Bits"."Day/Night Transition Bit" := 1; END_IF;
END_REGION
END_FUNCTION_BLOCK

FUNCTION_BLOCK "Get Weather Station Data"   // FB13, LAD
{ S7_Optimized_Access := 'TRUE' }
VERSION : 0.1
   VAR
      MBTO : Bool;
      OS3 : Bool;
   END_VAR
   VAR_TEMP
      temp_int : Byte;
      calc_out : Int;
   END_VAR
   VAR_TEMP   // added for the SCL form of the ladder/FBD networks
      _w1 : Bool;
      _w2 : Bool;
      _w3 : Bool;
   END_VAR
BEGIN

REGION Network 1
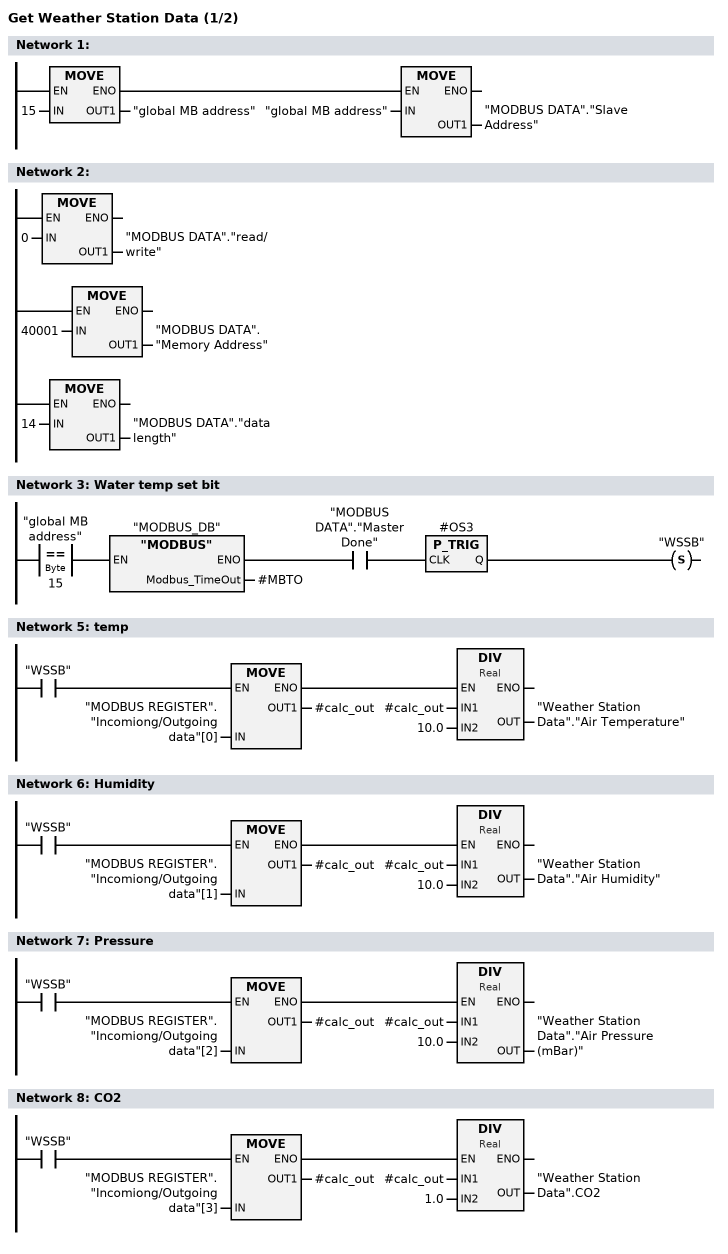
   RUNG wire#powerrail
      Move(in := 15, out1 => "global MB address")
      Move(in := "global MB address", out1 => "MODBUS DATA"."Slave Address")
   END_RUNG
   // the same network as SCL:
   "global MB address" := 15;
   "MODBUS DATA"."Slave Address" := "global MB address";
END_REGION

REGION Network 2
   RUNG wire#powerrail
      Move(in := 0, out1 => "MODBUS DATA"."read/write")
   END_RUNG
   RUNG wire#powerrail
      Move(in := 40001, out1 => "MODBUS DATA"."Memory Address")
   END_RUNG
   RUNG wire#powerrail
      Move(in := 14, out1 => "MODBUS DATA"."data length")
   END_RUNG
   // the same network as SCL:
   "MODBUS DATA"."read/write" := 0;
   "MODBUS DATA"."Memory Address" := 40001;
   "MODBUS DATA"."data length" := 14;
END_REGION

REGION Network 3: Water temp set bit
   RUNG wire#powerrail
      { S7_Templates := "SrcType := Byte" } EQ_Contact(in1 := "global MB address", in2 := 15)
      "MODBUS_DB"(Modbus_TimeOut => #MBTO)
      Contact( "MODBUS DATA"."Master Done" )
      P_Trig( #OS3 )
      S_Coil( "WSSB" )
   END_RUNG
   // the same network as SCL:
   "MODBUS_DB"(EN := "global MB address" = 15, Modbus_TimeOut => #MBTO, ENO => #_w1);   // "MODBUS"
   #_w2 := #_w1 AND "MODBUS DATA"."Master Done";
   #_w3 := #_w2 AND NOT #OS3;   // rising edge
   #OS3 := #_w2;
   IF #_w3 THEN "WSSB" := TRUE; END_IF;
END_REGION

REGION Network 5: temp
   RUNG wire#powerrail
      Contact( "WSSB" )
      Move(in := "MODBUS REGISTER"."Incomiong/Outgoing data"[0], out1 => #calc_out)
      { S7_Templates := "SrcType := Real" } Div(in1 := #calc_out, in2 := 10.0, out => "Weather Station Data"."Air Temperature")
   END_RUNG
   // the same network as SCL:
   IF "WSSB" THEN
       #calc_out := "MODBUS REGISTER"."Incomiong/Outgoing data"[0];
       "Weather Station Data"."Air Temperature" := #calc_out / 10.0;
   END_IF;
END_REGION

REGION Network 6: Humidity
   RUNG wire#powerrail
      Contact( "WSSB" )
      Move(in := "MODBUS REGISTER"."Incomiong/Outgoing data"[1], out1 => #calc_out)
      { S7_Templates := "SrcType := Real" } Div(in1 := #calc_out, in2 := 10.0, out => "Weather Station Data"."Air Humidity")
   END_RUNG
   // the same network as SCL:
   IF "WSSB" THEN
       #calc_out := "MODBUS REGISTER"."Incomiong/Outgoing data"[1];
       "Weather Station Data"."Air Humidity" := #calc_out / 10.0;
   END_IF;
END_REGION

REGION Network 7: Pressure
   RUNG wire#powerrail
      Contact( "WSSB" )
      Move(in := "MODBUS REGISTER"."Incomiong/Outgoing data"[2], out1 => #calc_out)
      { S7_Templates := "SrcType := Real" } Div(in1 := #calc_out, in2 := 10.0, out => "Weather Station Data"."Air Pressure (mBar)")
   END_RUNG
   // the same network as SCL:
   IF "WSSB" THEN
       #calc_out := "MODBUS REGISTER"."Incomiong/Outgoing data"[2];
       "Weather Station Data"."Air Pressure (mBar)" := #calc_out / 10.0;
   END_IF;
END_REGION

REGION Network 8: CO2
   RUNG wire#powerrail
      Contact( "WSSB" )
      Move(in := "MODBUS REGISTER"."Incomiong/Outgoing data"[3], out1 => #calc_out)
      { S7_Templates := "SrcType := Real" } Div(in1 := #calc_out, in2 := 1.0, out => "Weather Station Data".CO2)
   END_RUNG
   // the same network as SCL:
   IF "WSSB" THEN
       #calc_out := "MODBUS REGISTER"."Incomiong/Outgoing data"[3];
       "Weather Station Data".CO2 := #calc_out / 1.0;
   END_IF;
END_REGION

REGION Network 9: PM 2.5
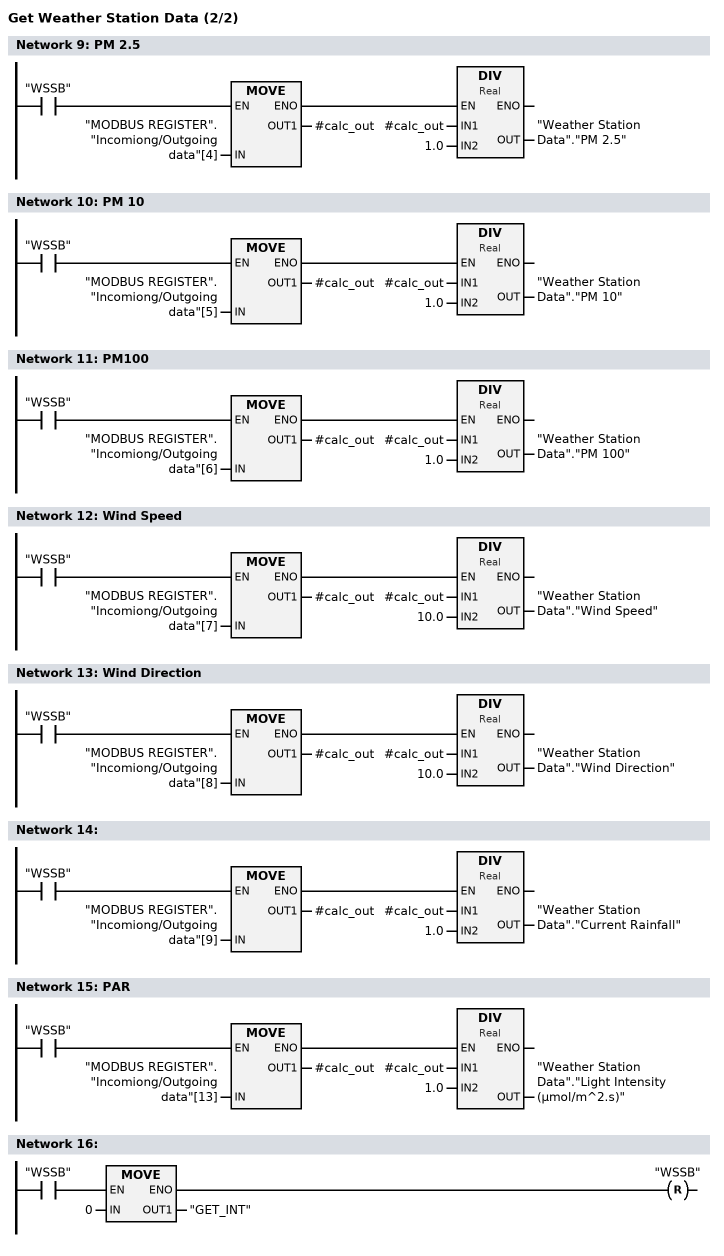
   RUNG wire#powerrail
      Contact( "WSSB" )
      Move(in := "MODBUS REGISTER"."Incomiong/Outgoing data"[4], out1 => #calc_out)
      { S7_Templates := "SrcType := Real" } Div(in1 := #calc_out, in2 := 1.0, out => "Weather Station Data"."PM 2.5")
   END_RUNG
   // the same network as SCL:
   IF "WSSB" THEN
       #calc_out := "MODBUS REGISTER"."Incomiong/Outgoing data"[4];
       "Weather Station Data"."PM 2.5" := #calc_out / 1.0;
   END_IF;
END_REGION

REGION Network 10: PM 10
   RUNG wire#powerrail
      Contact( "WSSB" )
      Move(in := "MODBUS REGISTER"."Incomiong/Outgoing data"[5], out1 => #calc_out)
      { S7_Templates := "SrcType := Real" } Div(in1 := #calc_out, in2 := 1.0, out => "Weather Station Data"."PM 10")
   END_RUNG
   // the same network as SCL:
   IF "WSSB" THEN
       #calc_out := "MODBUS REGISTER"."Incomiong/Outgoing data"[5];
       "Weather Station Data"."PM 10" := #calc_out / 1.0;
   END_IF;
END_REGION

REGION Network 11: PM100
   RUNG wire#powerrail
      Contact( "WSSB" )
      Move(in := "MODBUS REGISTER"."Incomiong/Outgoing data"[6], out1 => #calc_out)
      { S7_Templates := "SrcType := Real" } Div(in1 := #calc_out, in2 := 1.0, out => "Weather Station Data"."PM 100")
   END_RUNG
   // the same network as SCL:
   IF "WSSB" THEN
       #calc_out := "MODBUS REGISTER"."Incomiong/Outgoing data"[6];
       "Weather Station Data"."PM 100" := #calc_out / 1.0;
   END_IF;
END_REGION

REGION Network 12: Wind Speed
   RUNG wire#powerrail
      Contact( "WSSB" )
      Move(in := "MODBUS REGISTER"."Incomiong/Outgoing data"[7], out1 => #calc_out)
      { S7_Templates := "SrcType := Real" } Div(in1 := #calc_out, in2 := 10.0, out => "Weather Station Data"."Wind Speed")
   END_RUNG
   // the same network as SCL:
   IF "WSSB" THEN
       #calc_out := "MODBUS REGISTER"."Incomiong/Outgoing data"[7];
       "Weather Station Data"."Wind Speed" := #calc_out / 10.0;
   END_IF;
END_REGION

REGION Network 13: Wind Direction
   RUNG wire#powerrail
      Contact( "WSSB" )
      Move(in := "MODBUS REGISTER"."Incomiong/Outgoing data"[8], out1 => #calc_out)
      { S7_Templates := "SrcType := Real" } Div(in1 := #calc_out, in2 := 10.0, out => "Weather Station Data"."Wind Direction")
   END_RUNG
   // the same network as SCL:
   IF "WSSB" THEN
       #calc_out := "MODBUS REGISTER"."Incomiong/Outgoing data"[8];
       "Weather Station Data"."Wind Direction" := #calc_out / 10.0;
   END_IF;
END_REGION

REGION Network 14
   RUNG wire#powerrail
      Contact( "WSSB" )
      Move(in := "MODBUS REGISTER"."Incomiong/Outgoing data"[9], out1 => #calc_out)
      { S7_Templates := "SrcType := Real" } Div(in1 := #calc_out, in2 := 1.0, out => "Weather Station Data"."Current Rainfall")
   END_RUNG
   // the same network as SCL:
   IF "WSSB" THEN
       #calc_out := "MODBUS REGISTER"."Incomiong/Outgoing data"[9];
       "Weather Station Data"."Current Rainfall" := #calc_out / 1.0;
   END_IF;
END_REGION

REGION Network 15: PAR
   RUNG wire#powerrail
      Contact( "WSSB" )
      Move(in := "MODBUS REGISTER"."Incomiong/Outgoing data"[13], out1 => #calc_out)
      { S7_Templates := "SrcType := Real" } Div(in1 := #calc_out, in2 := 1.0, out => "Weather Station Data"."Light Intensity (μmol/m^2.s)")
   END_RUNG
   // the same network as SCL:
   IF "WSSB" THEN
       #calc_out := "MODBUS REGISTER"."Incomiong/Outgoing data"[13];
       "Weather Station Data"."Light Intensity (μmol/m^2.s)" := #calc_out / 1.0;
   END_IF;
END_REGION

REGION Network 16
   RUNG wire#powerrail
      Contact( "WSSB" )
      Move(in := 0, out1 => "GET_INT")
      R_Coil( "WSSB" )
   END_RUNG
   // the same network as SCL:
   IF "WSSB" THEN
       "GET_INT" := 0;
       "WSSB" := FALSE;
   END_IF;
END_REGION
END_FUNCTION_BLOCK

FUNCTION_BLOCK "Emergency_Stop"   // FB14, LAD
TITLE = Emergency stop routine
{ S7_Optimized_Access := 'TRUE' }
AUTHOR : FF
VERSION : 0.1
// Includes Estop buttons and any safety flags such as malfunction in one of the fans/pumps
   VAR_TEMP   // added for the SCL form of the ladder/FBD networks
      _w1 : Bool;
   END_VAR
BEGIN

REGION Network 1
   // Estop on the panel monitoring
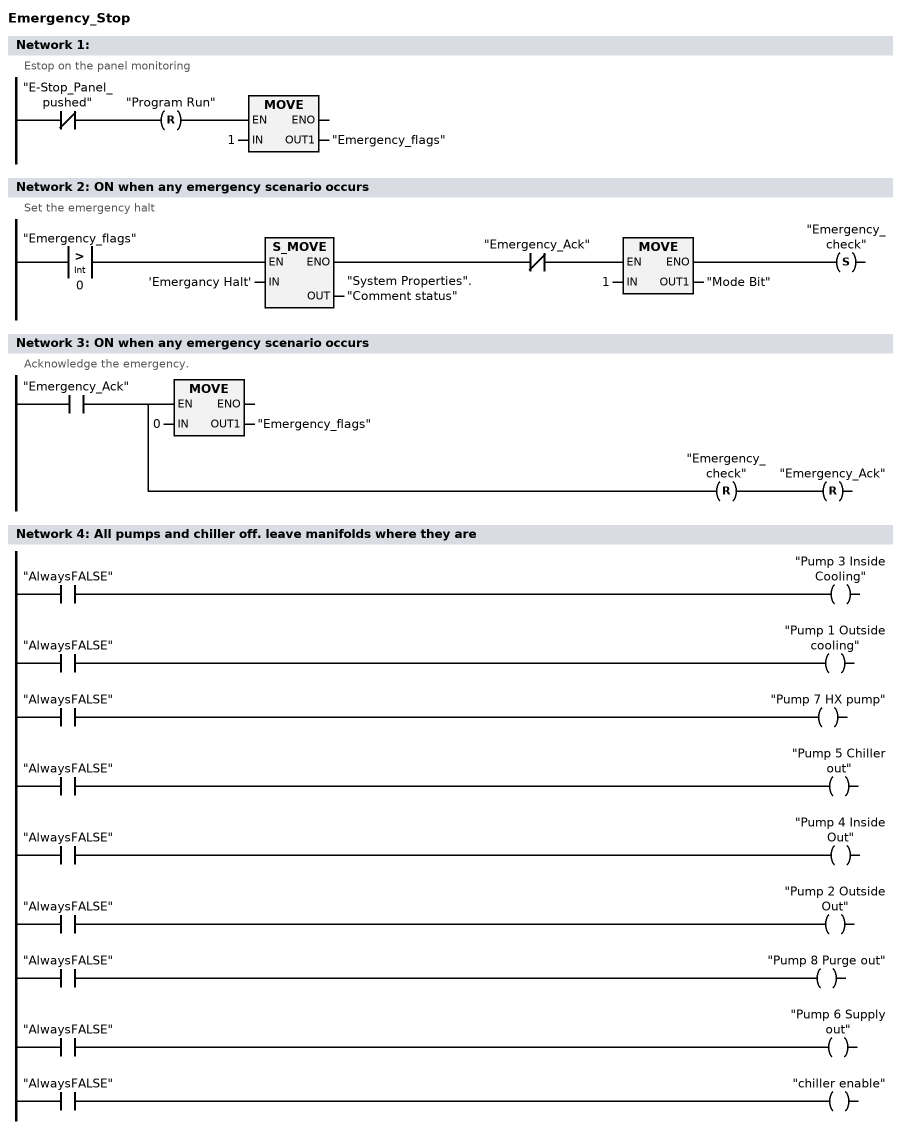
   RUNG wire#powerrail
      I_Contact( "E-Stop_Panel_pushed" )
      R_Coil( "Program Run" )
      Move(in := 1, out1 => "Emergency_flags")
   END_RUNG
   // the same network as SCL:
   IF NOT "E-Stop_Panel_pushed" THEN
       "Program Run" := FALSE;
       "Emergency_flags" := 1;
   END_IF;
END_REGION

REGION Network 2: ON when any emergency scenario occurs
   // Set the emergency halt
   RUNG wire#powerrail
      { S7_Templates := "SrcType := Int" } GT_Contact(in1 := "Emergency_flags", in2 := 0)
      S_Move(in := 'Emergancy Halt', out => "System Properties"."Comment status")
      I_Contact( "Emergency_Ack" )
      Move(in := 1, out1 => "Mode Bit")
      S_Coil( "Emergency_check" )
   END_RUNG
   // the same network as SCL:
   #_w1 := "Emergency_flags" > 0;
   IF #_w1 THEN "System Properties"."Comment status" := 'Emergancy Halt'; END_IF;
   IF #_w1 AND NOT "Emergency_Ack" THEN
       "Mode Bit" := 1;
       "Emergency_check" := TRUE;
   END_IF;
END_REGION

REGION Network 3: ON when any emergency scenario occurs
   // Acknowledge the emergency.
   RUNG wire#powerrail
      Contact( "Emergency_Ack" )
      wire#w1
      Move(in := 0, out1 => "Emergency_flags")
   END_RUNG
   RUNG wire#w1
      R_Coil( "Emergency_check" )
      R_Coil( "Emergency_Ack" )
   END_RUNG
   // the same network as SCL:
   IF "Emergency_Ack" THEN
       "Emergency_flags" := 0;
       "Emergency_check" := FALSE;
       "Emergency_Ack" := FALSE;
   END_IF;
END_REGION

REGION Network 4: All pumps and chiller off. leave manifolds where they are
   RUNG wire#powerrail
      Contact( "AlwaysFALSE" )
      Coil( "Pump 3 Inside Cooling" )
   END_RUNG
   RUNG wire#powerrail
      Contact( "AlwaysFALSE" )
      Coil( "Pump 1 Outside cooling" )
   END_RUNG
   RUNG wire#powerrail
      Contact( "AlwaysFALSE" )
      Coil( "Pump 7 HX pump" )
   END_RUNG
   RUNG wire#powerrail
      Contact( "AlwaysFALSE" )
      Coil( "Pump 5 Chiller out" )
   END_RUNG
   RUNG wire#powerrail
      Contact( "AlwaysFALSE" )
      Coil( "Pump 4 Inside Out" )
   END_RUNG
   RUNG wire#powerrail
      Contact( "AlwaysFALSE" )
      Coil( "Pump 2 Outside Out" )
   END_RUNG
   RUNG wire#powerrail
      Contact( "AlwaysFALSE" )
      Coil( "Pump 8 Purge out" )
   END_RUNG
   RUNG wire#powerrail
      Contact( "AlwaysFALSE" )
      Coil( "Pump 6 Supply out" )
   END_RUNG
   RUNG wire#powerrail
      Contact( "AlwaysFALSE" )
      Coil( "chiller enable" )
   END_RUNG
   // the same network as SCL:
   "Pump 3 Inside Cooling" := "AlwaysFALSE";
   "Pump 1 Outside cooling" := "AlwaysFALSE";
   "Pump 7 HX pump" := "AlwaysFALSE";
   "Pump 5 Chiller out" := "AlwaysFALSE";
   "Pump 4 Inside Out" := "AlwaysFALSE";
   "Pump 2 Outside Out" := "AlwaysFALSE";
   "Pump 8 Purge out" := "AlwaysFALSE";
   "Pump 6 Supply out" := "AlwaysFALSE";
   "chiller enable" := "AlwaysFALSE";
END_REGION
END_FUNCTION_BLOCK

FUNCTION_BLOCK "MODBUS"   // FB15, LAD
{ S7_Optimized_Access := 'TRUE' }
VERSION : 0.1
   VAR_OUTPUT
      Modbus_TimeOut : Bool;
   END_VAR
   VAR
      resetTime : Bool;
      OS3 : Bool;
   END_VAR
   VAR_TEMP
      OS1 : Bool;
      temp : Bool;
      resetT : Bool;
      OS2 : Bool;
   END_VAR
   VAR_TEMP   // added for the SCL form of the ladder/FBD networks
      _w1 : Bool;
   END_VAR
BEGIN

REGION Network 1
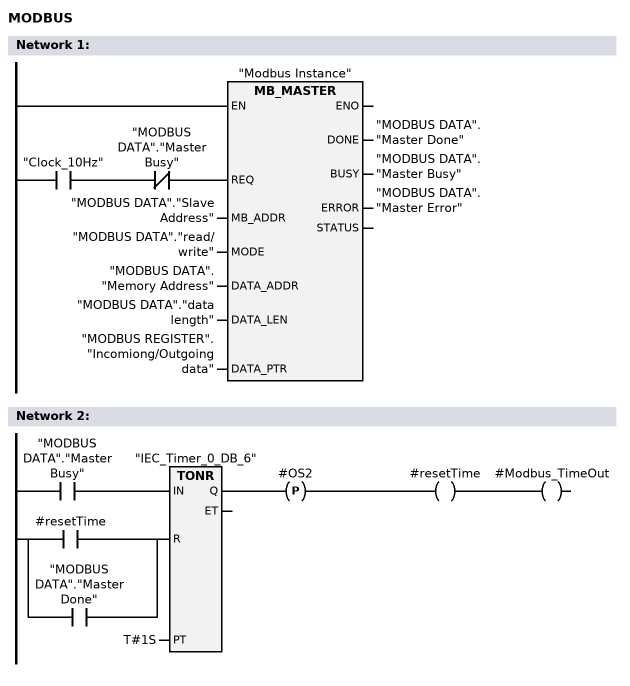
   "Modbus Instance"(REQ := "Clock_10Hz" AND NOT "MODBUS DATA"."Master Busy",   // MB_MASTER
                     MB_ADDR := "MODBUS DATA"."Slave Address",
                     MODE := "MODBUS DATA"."read/write",
                     DATA_ADDR := "MODBUS DATA"."Memory Address",
                     DATA_LEN := "MODBUS DATA"."data length",
                     DATA_PTR := "MODBUS REGISTER"."Incomiong/Outgoing data",
                     DONE => "MODBUS DATA"."Master Done",
                     BUSY => "MODBUS DATA"."Master Busy",
                     ERROR => "MODBUS DATA"."Master Error");
END_REGION

REGION Network 2
   "IEC_Timer_0_DB_6".TONR(IN := "MODBUS DATA"."Master Busy",
                           R := #resetTime OR "MODBUS DATA"."Master Done",
                           PT := T#1S);
   #_w1 := "IEC_Timer_0_DB_6".Q AND NOT #OS2;   // rising edge
   #OS2 := "IEC_Timer_0_DB_6".Q;
   #resetTime := #_w1;
   #Modbus_TimeOut := #_w1;
END_REGION
END_FUNCTION_BLOCK

FUNCTION_BLOCK "Get Ts and Hs"   // FB16, LAD
{ S7_Optimized_Access := 'TRUE' }
VERSION : 0.1
   VAR
      Raw_1 : Int;
      dev_1 : Real;
      Raw_2 : Int;
      dev_2 : Real;
      MBTO : Bool;
      OS7 : Bool;
      OS6 : Bool;
      OS8 : Bool;
      OS9 : Bool;
   END_VAR
   VAR_TEMP
      OS2 : Bool;
      OS3 : Bool;
      OS4 : Bool;
      OS5 : Bool;
      MBTO1 : Bool;
      MBTO2 : Bool;
      MBTO3 : Bool;
   END_VAR
   VAR_TEMP   // added for the SCL form of the ladder/FBD networks
      _w1 : Bool;
      _w2 : Bool;
      _w3 : Bool;
      _w4 : Bool;
   END_VAR
BEGIN

REGION Network 1
   // address;
   // 20 - Ambient
   // 21 - GH
   // 22 - Output of outside rig
   // 23 - Output of Inside rig
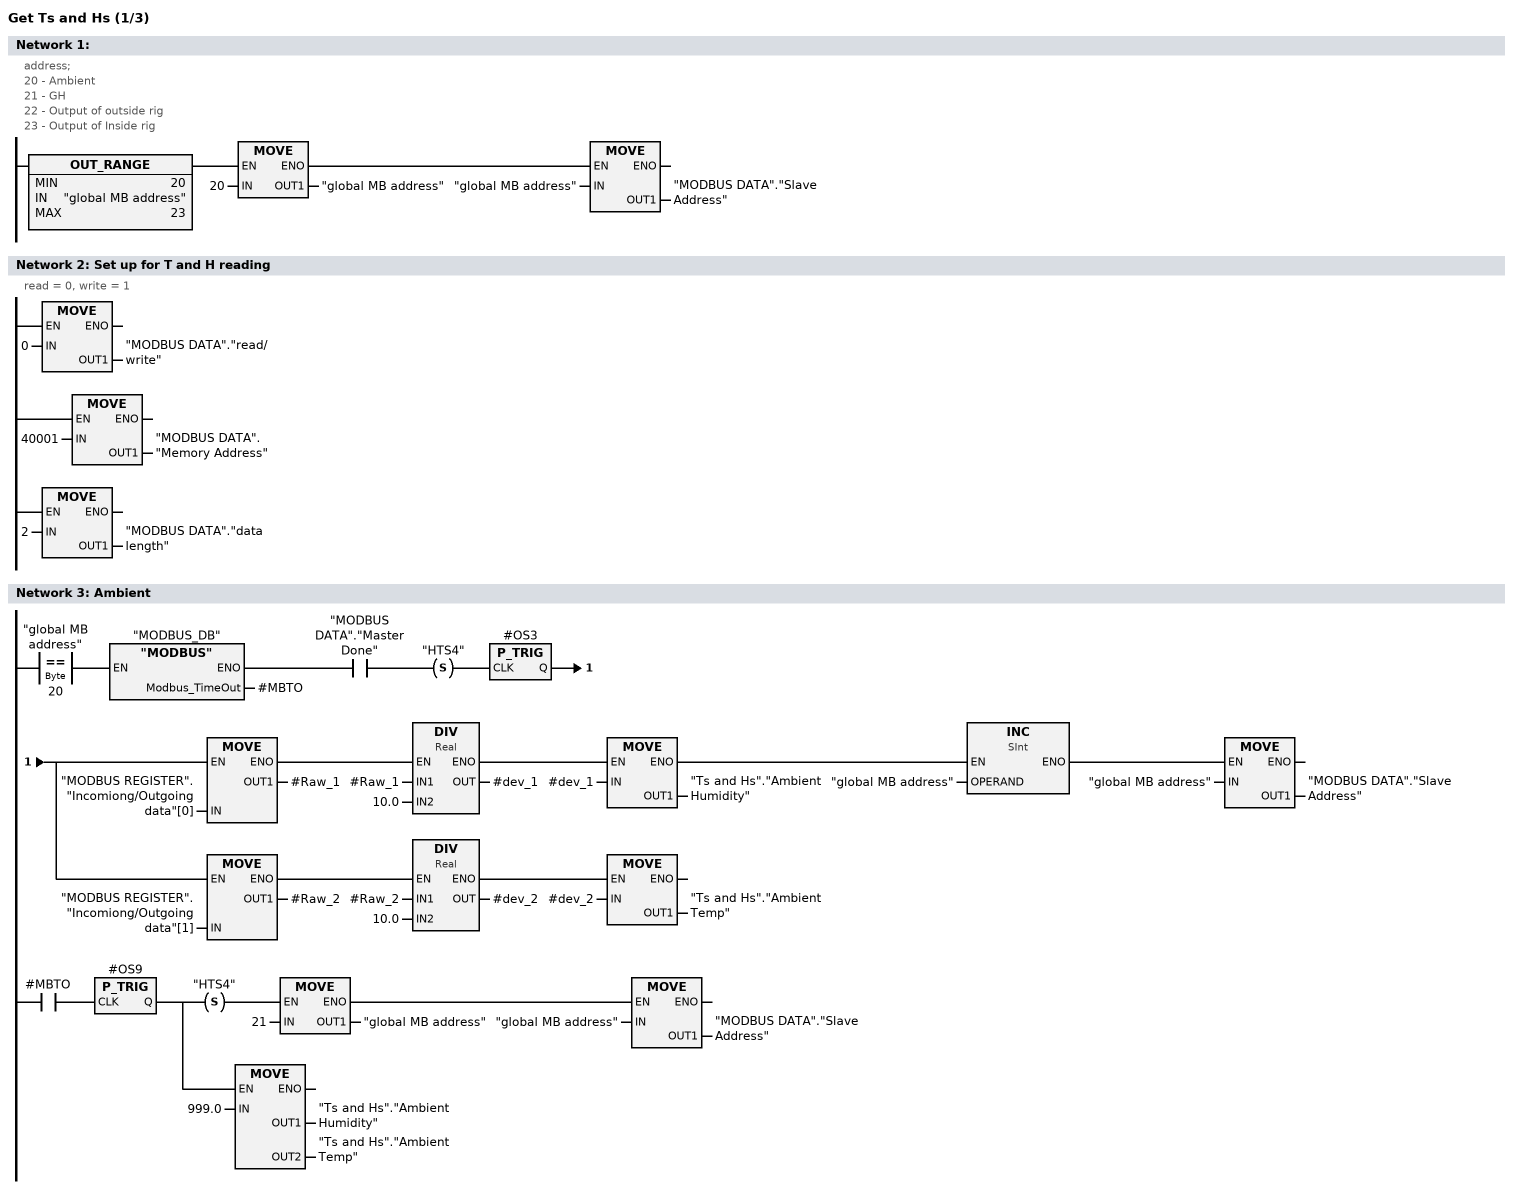
   #_w1 := ("global MB address" < 20) OR ("global MB address" > 23);
   IF #_w1 THEN
       "global MB address" := 20;
       "MODBUS DATA"."Slave Address" := "global MB address";
   END_IF;
END_REGION

REGION Network 2: Set up for T and H reading
   // read = 0, write = 1
   RUNG wire#powerrail
      Move(in := 0, out1 => "MODBUS DATA"."read/write")
   END_RUNG
   RUNG wire#powerrail
      Move(in := 40001, out1 => "MODBUS DATA"."Memory Address")
   END_RUNG
   RUNG wire#powerrail
      Move(in := 2, out1 => "MODBUS DATA"."data length")
   END_RUNG
   // the same network as SCL:
   "MODBUS DATA"."read/write" := 0;
   "MODBUS DATA"."Memory Address" := 40001;
   "MODBUS DATA"."data length" := 2;
END_REGION

REGION Network 3: Ambient
   RUNG wire#powerrail
      { S7_Templates := "SrcType := Byte" } EQ_Contact(in1 := "global MB address", in2 := 20)
      "MODBUS_DB"(Modbus_TimeOut => #MBTO)
      Contact( "MODBUS DATA"."Master Done" )
      S_Coil( "HTS4" )
      P_Trig( #OS3 )
      wire#w1
      Move(in := "MODBUS REGISTER"."Incomiong/Outgoing data"[0], out1 => #Raw_1)
      { S7_Templates := "SrcType := Real" } Div(in1 := #Raw_1, in2 := 10.0, out => #dev_1)
      Move(in := #dev_1, out1 => "Ts and Hs"."Ambient Humidity")
      { S7_Templates := "DestType := SInt" } Inc( "global MB address" )
      Move(in := "global MB address", out1 => "MODBUS DATA"."Slave Address")
   END_RUNG
   RUNG wire#w1
      Move(in := "MODBUS REGISTER"."Incomiong/Outgoing data"[1], out1 => #Raw_2)
      { S7_Templates := "SrcType := Real" } Div(in1 := #Raw_2, in2 := 10.0, out => #dev_2)
      Move(in := #dev_2, out1 => "Ts and Hs"."Ambient Temp")
   END_RUNG
   RUNG wire#powerrail
      Contact( #MBTO )
      P_Trig( #OS9 )
      wire#w2
      S_Coil( "HTS4" )
      Move(in := 21, out1 => "global MB address")
      Move(in := "global MB address", out1 => "MODBUS DATA"."Slave Address")
   END_RUNG
   RUNG wire#w2
      Move(in := 999.0, out1 => "Ts and Hs"."Ambient Humidity", out2 => "Ts and Hs"."Ambient Temp")
   END_RUNG
   // the same network as SCL:
   "MODBUS_DB"(EN := "global MB address" = 20, Modbus_TimeOut => #MBTO, ENO => #_w1);   // "MODBUS"
   #_w2 := #_w1 AND "MODBUS DATA"."Master Done";
   IF #_w2 THEN "HTS4" := TRUE; END_IF;
   #_w3 := #_w2 AND NOT #OS3;   // rising edge
   #OS3 := #_w2;
   IF #_w3 THEN
       #Raw_1 := "MODBUS REGISTER"."Incomiong/Outgoing data"[0];
       #dev_1 := #Raw_1 / 10.0;
       "Ts and Hs"."Ambient Humidity" := #dev_1;
       "global MB address" := "global MB address" + 1;
       "MODBUS DATA"."Slave Address" := "global MB address";
       #Raw_2 := "MODBUS REGISTER"."Incomiong/Outgoing data"[1];
       #dev_2 := #Raw_2 / 10.0;
       "Ts and Hs"."Ambient Temp" := #dev_2;
   END_IF;
   #_w4 := #MBTO AND NOT #OS9;   // rising edge
   #OS9 := #MBTO;
   IF #_w4 THEN
       "HTS4" := TRUE;
       "global MB address" := 21;
       "MODBUS DATA"."Slave Address" := "global MB address";
       "Ts and Hs"."Ambient Humidity" := 999.0;
       "Ts and Hs"."Ambient Temp" := 999.0;
   END_IF;
END_REGION

REGION Network 4: Greenhouse
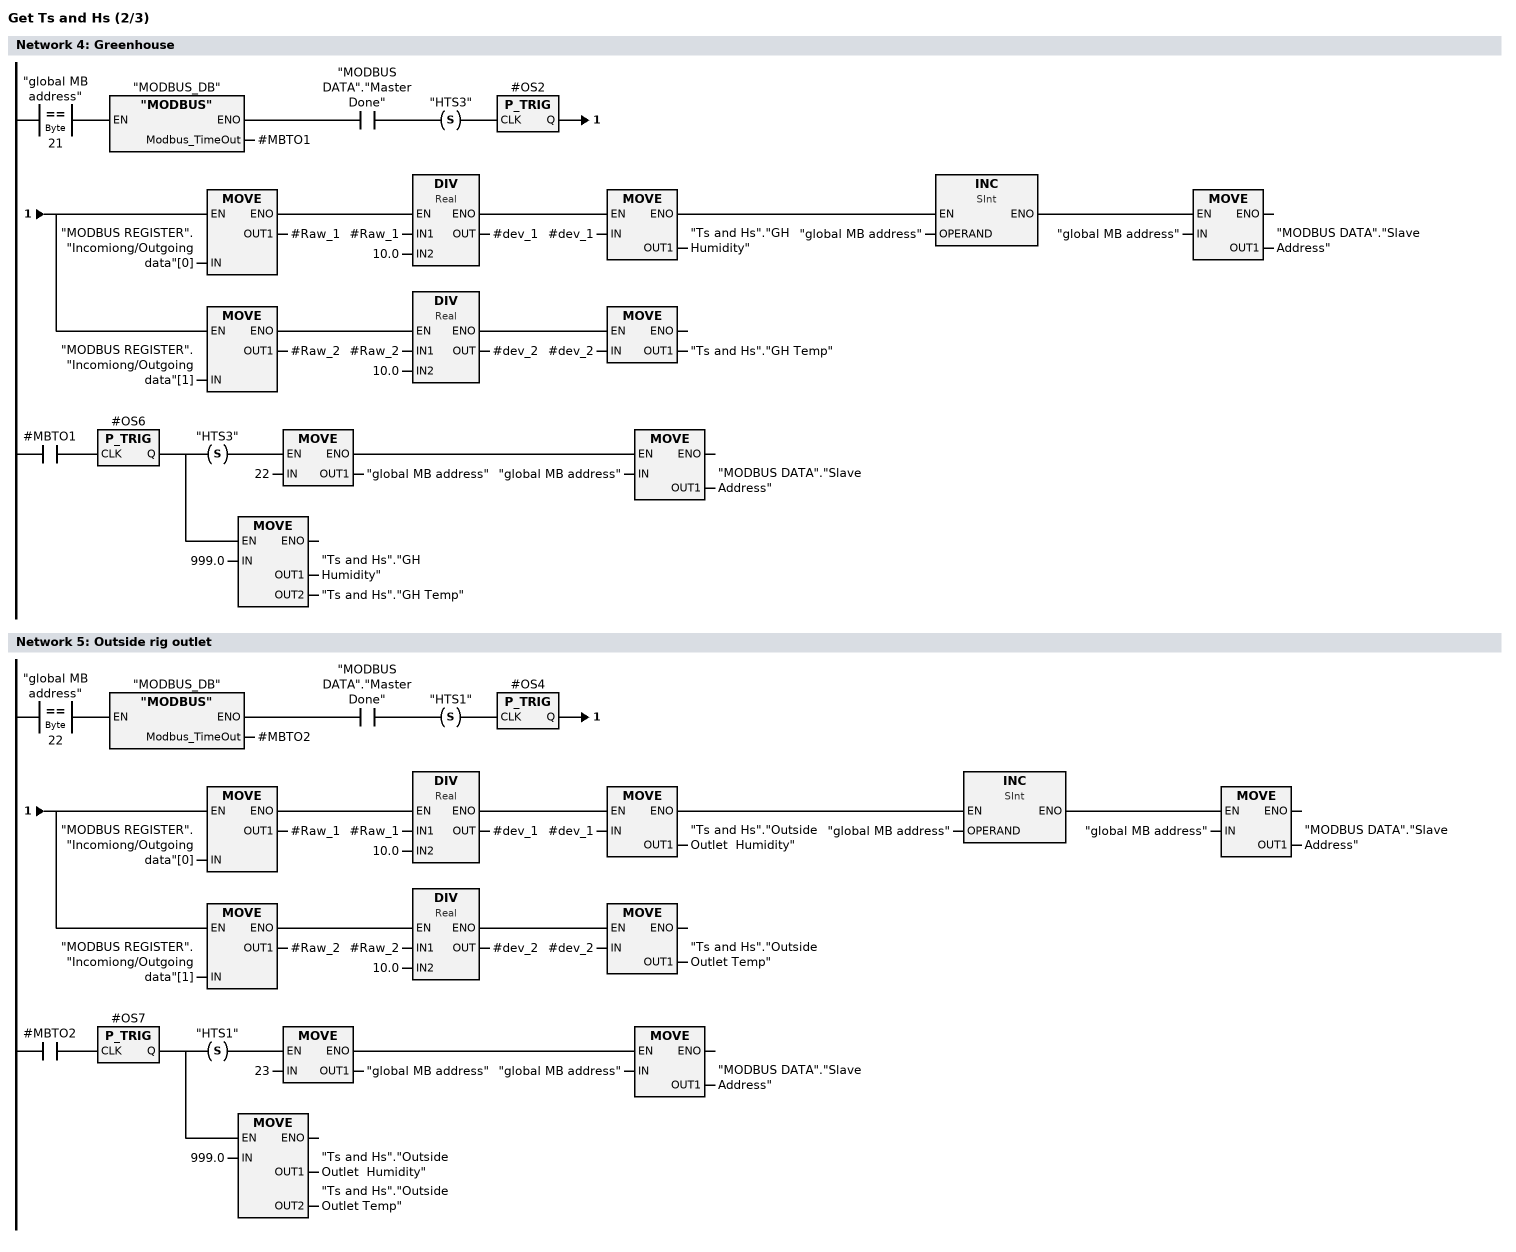
   RUNG wire#powerrail
      { S7_Templates := "SrcType := Byte" } EQ_Contact(in1 := "global MB address", in2 := 21)
      "MODBUS_DB"(Modbus_TimeOut => #MBTO1)
      Contact( "MODBUS DATA"."Master Done" )
      S_Coil( "HTS3" )
      P_Trig( #OS2 )
      wire#w1
      Move(in := "MODBUS REGISTER"."Incomiong/Outgoing data"[0], out1 => #Raw_1)
      { S7_Templates := "SrcType := Real" } Div(in1 := #Raw_1, in2 := 10.0, out => #dev_1)
      Move(in := #dev_1, out1 => "Ts and Hs"."GH Humidity")
      { S7_Templates := "DestType := SInt" } Inc( "global MB address" )
      Move(in := "global MB address", out1 => "MODBUS DATA"."Slave Address")
   END_RUNG
   RUNG wire#w1
      Move(in := "MODBUS REGISTER"."Incomiong/Outgoing data"[1], out1 => #Raw_2)
      { S7_Templates := "SrcType := Real" } Div(in1 := #Raw_2, in2 := 10.0, out => #dev_2)
      Move(in := #dev_2, out1 => "Ts and Hs"."GH Temp")
   END_RUNG
   RUNG wire#powerrail
      Contact( #MBTO1 )
      P_Trig( #OS6 )
      wire#w2
      S_Coil( "HTS3" )
      Move(in := 22, out1 => "global MB address")
      Move(in := "global MB address", out1 => "MODBUS DATA"."Slave Address")
   END_RUNG
   RUNG wire#w2
      Move(in := 999.0, out1 => "Ts and Hs"."GH Humidity", out2 => "Ts and Hs"."GH Temp")
   END_RUNG
   // the same network as SCL:
   "MODBUS_DB"(EN := "global MB address" = 21, Modbus_TimeOut => #MBTO1, ENO => #_w1);   // "MODBUS"
   #_w2 := #_w1 AND "MODBUS DATA"."Master Done";
   IF #_w2 THEN "HTS3" := TRUE; END_IF;
   #_w3 := #_w2 AND NOT #OS2;   // rising edge
   #OS2 := #_w2;
   IF #_w3 THEN
       #Raw_1 := "MODBUS REGISTER"."Incomiong/Outgoing data"[0];
       #dev_1 := #Raw_1 / 10.0;
       "Ts and Hs"."GH Humidity" := #dev_1;
       "global MB address" := "global MB address" + 1;
       "MODBUS DATA"."Slave Address" := "global MB address";
       #Raw_2 := "MODBUS REGISTER"."Incomiong/Outgoing data"[1];
       #dev_2 := #Raw_2 / 10.0;
       "Ts and Hs"."GH Temp" := #dev_2;
   END_IF;
   #_w4 := #MBTO1 AND NOT #OS6;   // rising edge
   #OS6 := #MBTO1;
   IF #_w4 THEN
       "HTS3" := TRUE;
       "global MB address" := 22;
       "MODBUS DATA"."Slave Address" := "global MB address";
       "Ts and Hs"."GH Humidity" := 999.0;
       "Ts and Hs"."GH Temp" := 999.0;
   END_IF;
END_REGION

REGION Network 5: Outside rig outlet
   RUNG wire#powerrail
      { S7_Templates := "SrcType := Byte" } EQ_Contact(in1 := "global MB address", in2 := 22)
      "MODBUS_DB"(Modbus_TimeOut => #MBTO2)
      Contact( "MODBUS DATA"."Master Done" )
      S_Coil( "HTS1" )
      P_Trig( #OS4 )
      wire#w1
      Move(in := "MODBUS REGISTER"."Incomiong/Outgoing data"[0], out1 => #Raw_1)
      { S7_Templates := "SrcType := Real" } Div(in1 := #Raw_1, in2 := 10.0, out => #dev_1)
      Move(in := #dev_1, out1 => "Ts and Hs"."Outside Outlet  Humidity")
      { S7_Templates := "DestType := SInt" } Inc( "global MB address" )
      Move(in := "global MB address", out1 => "MODBUS DATA"."Slave Address")
   END_RUNG
   RUNG wire#w1
      Move(in := "MODBUS REGISTER"."Incomiong/Outgoing data"[1], out1 => #Raw_2)
      { S7_Templates := "SrcType := Real" } Div(in1 := #Raw_2, in2 := 10.0, out => #dev_2)
      Move(in := #dev_2, out1 => "Ts and Hs"."Outside Outlet Temp")
   END_RUNG
   RUNG wire#powerrail
      Contact( #MBTO2 )
      P_Trig( #OS7 )
      wire#w2
      S_Coil( "HTS1" )
      Move(in := 23, out1 => "global MB address")
      Move(in := "global MB address", out1 => "MODBUS DATA"."Slave Address")
   END_RUNG
   RUNG wire#w2
      Move(in := 999.0, out1 => "Ts and Hs"."Outside Outlet  Humidity", out2 => "Ts and Hs"."Outside Outlet Temp")
   END_RUNG
   // the same network as SCL:
   "MODBUS_DB"(EN := "global MB address" = 22, Modbus_TimeOut => #MBTO2, ENO => #_w1);   // "MODBUS"
   #_w2 := #_w1 AND "MODBUS DATA"."Master Done";
   IF #_w2 THEN "HTS1" := TRUE; END_IF;
   #_w3 := #_w2 AND NOT #OS4;   // rising edge
   #OS4 := #_w2;
   IF #_w3 THEN
       #Raw_1 := "MODBUS REGISTER"."Incomiong/Outgoing data"[0];
       #dev_1 := #Raw_1 / 10.0;
       "Ts and Hs"."Outside Outlet  Humidity" := #dev_1;
       "global MB address" := "global MB address" + 1;
       "MODBUS DATA"."Slave Address" := "global MB address";
       #Raw_2 := "MODBUS REGISTER"."Incomiong/Outgoing data"[1];
       #dev_2 := #Raw_2 / 10.0;
       "Ts and Hs"."Outside Outlet Temp" := #dev_2;
   END_IF;
   #_w4 := #MBTO2 AND NOT #OS7;   // rising edge
   #OS7 := #MBTO2;
   IF #_w4 THEN
       "HTS1" := TRUE;
       "global MB address" := 23;
       "MODBUS DATA"."Slave Address" := "global MB address";
       "Ts and Hs"."Outside Outlet  Humidity" := 999.0;
       "Ts and Hs"."Outside Outlet Temp" := 999.0;
   END_IF;
END_REGION

REGION Network 6: Inside Rig Outlet
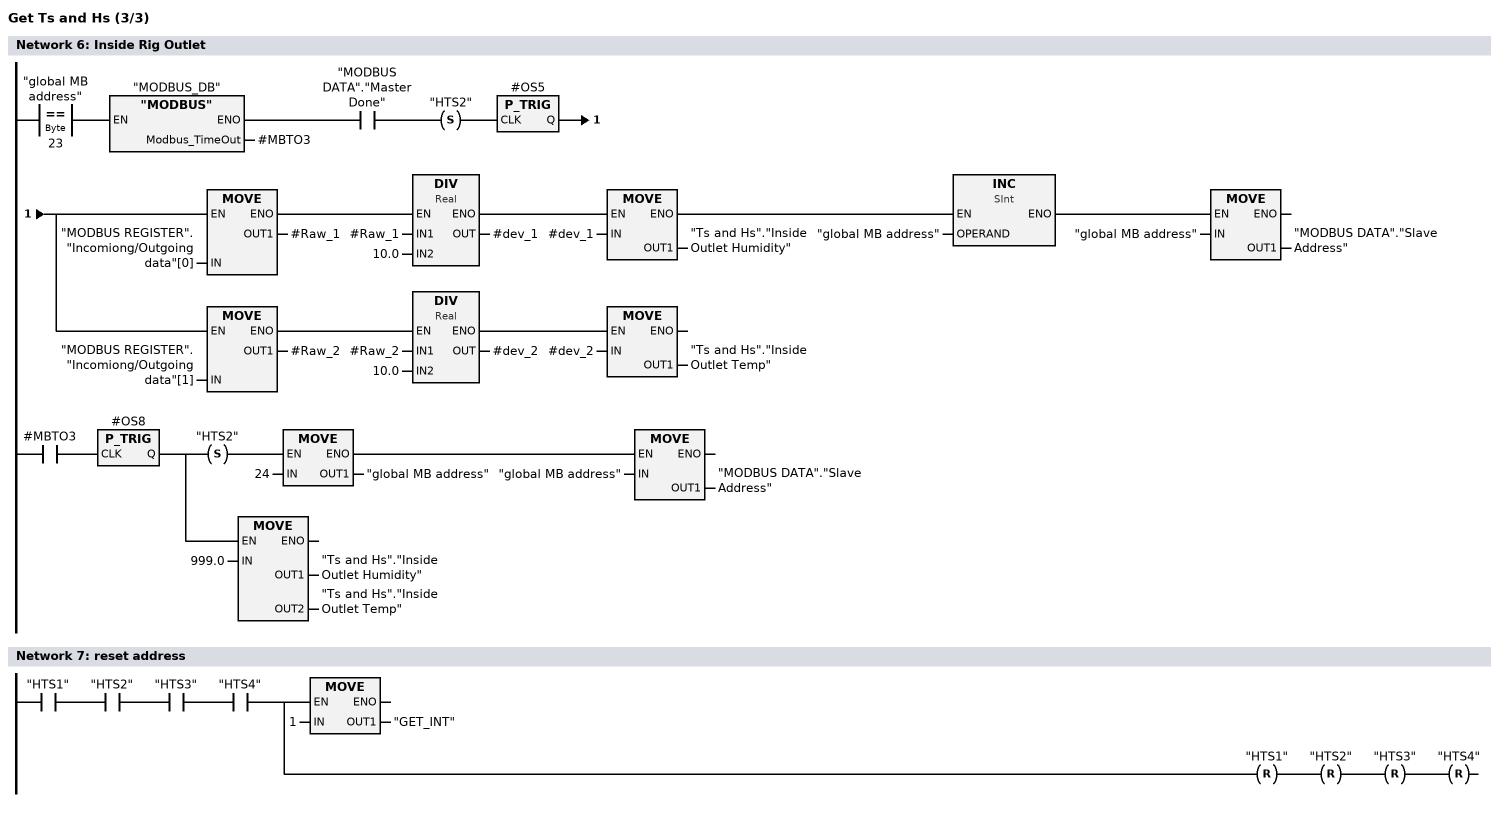
   RUNG wire#powerrail
      { S7_Templates := "SrcType := Byte" } EQ_Contact(in1 := "global MB address", in2 := 23)
      "MODBUS_DB"(Modbus_TimeOut => #MBTO3)
      Contact( "MODBUS DATA"."Master Done" )
      S_Coil( "HTS2" )
      P_Trig( #OS5 )
      wire#w1
      Move(in := "MODBUS REGISTER"."Incomiong/Outgoing data"[0], out1 => #Raw_1)
      { S7_Templates := "SrcType := Real" } Div(in1 := #Raw_1, in2 := 10.0, out => #dev_1)
      Move(in := #dev_1, out1 => "Ts and Hs"."Inside Outlet Humidity")
      { S7_Templates := "DestType := SInt" } Inc( "global MB address" )
      Move(in := "global MB address", out1 => "MODBUS DATA"."Slave Address")
   END_RUNG
   RUNG wire#w1
      Move(in := "MODBUS REGISTER"."Incomiong/Outgoing data"[1], out1 => #Raw_2)
      { S7_Templates := "SrcType := Real" } Div(in1 := #Raw_2, in2 := 10.0, out => #dev_2)
      Move(in := #dev_2, out1 => "Ts and Hs"."Inside Outlet Temp")
   END_RUNG
   RUNG wire#powerrail
      Contact( #MBTO3 )
      P_Trig( #OS8 )
      wire#w2
      S_Coil( "HTS2" )
      Move(in := 24, out1 => "global MB address")
      Move(in := "global MB address", out1 => "MODBUS DATA"."Slave Address")
   END_RUNG
   RUNG wire#w2
      Move(in := 999.0, out1 => "Ts and Hs"."Inside Outlet Humidity", out2 => "Ts and Hs"."Inside Outlet Temp")
   END_RUNG
   // the same network as SCL:
   "MODBUS_DB"(EN := "global MB address" = 23, Modbus_TimeOut => #MBTO3, ENO => #_w1);   // "MODBUS"
   #_w2 := #_w1 AND "MODBUS DATA"."Master Done";
   IF #_w2 THEN "HTS2" := TRUE; END_IF;
   #_w3 := #_w2 AND NOT #OS5;   // rising edge
   #OS5 := #_w2;
   IF #_w3 THEN
       #Raw_1 := "MODBUS REGISTER"."Incomiong/Outgoing data"[0];
       #dev_1 := #Raw_1 / 10.0;
       "Ts and Hs"."Inside Outlet Humidity" := #dev_1;
       "global MB address" := "global MB address" + 1;
       "MODBUS DATA"."Slave Address" := "global MB address";
       #Raw_2 := "MODBUS REGISTER"."Incomiong/Outgoing data"[1];
       #dev_2 := #Raw_2 / 10.0;
       "Ts and Hs"."Inside Outlet Temp" := #dev_2;
   END_IF;
   #_w4 := #MBTO3 AND NOT #OS8;   // rising edge
   #OS8 := #MBTO3;
   IF #_w4 THEN
       "HTS2" := TRUE;
       "global MB address" := 24;
       "MODBUS DATA"."Slave Address" := "global MB address";
       "Ts and Hs"."Inside Outlet Humidity" := 999.0;
       "Ts and Hs"."Inside Outlet Temp" := 999.0;
   END_IF;
END_REGION

REGION Network 7: reset address
   RUNG wire#powerrail
      Contact( "HTS1" )
      Contact( "HTS2" )
      Contact( "HTS3" )
      Contact( "HTS4" )
      wire#w1
      Move(in := 1, out1 => "GET_INT")
   END_RUNG
   RUNG wire#w1
      R_Coil( "HTS1" )
      R_Coil( "HTS2" )
      R_Coil( "HTS3" )
      R_Coil( "HTS4" )
   END_RUNG
   // the same network as SCL:
   IF "HTS1" AND "HTS2" AND "HTS3" AND "HTS4" THEN "GET_INT" := 1; END_IF;
   #_w1 := "HTS1" AND "HTS2" AND "HTS3" AND "HTS4";
   IF #_w1 THEN
       "HTS1" := FALSE;
       "HTS2" := FALSE;
       "HTS3" := FALSE;
       "HTS4" := FALSE;
   END_IF;
END_REGION
END_FUNCTION_BLOCK

FUNCTION_BLOCK "Get Depths"   // FB17, LAD
{ S7_Optimized_Access := 'TRUE' }
VERSION : 0.1
   VAR
      Raw_1 : Int;
      dev_1 : Real;
      Raw_2 : Int;
      dev_2 : Real;
      MBTO : Bool;
      OS7 : Bool;
      OS6 : Bool;
      OS8 : Bool;
      OS9 : Bool;
   END_VAR
   VAR_TEMP
      OS2 : Bool;
      OS3 : Bool;
      OS4 : Bool;
      OS5 : Bool;
      MBTO1 : Bool;
      MBTO2 : Bool;
      MBTO3 : Bool;
   END_VAR
   VAR_TEMP   // added for the SCL form of the ladder/FBD networks
      _w1 : Bool;
      _w2 : Bool;
      _w3 : Bool;
      _w4 : Bool;
   END_VAR
BEGIN

REGION Network 1
   // address;
   // 20 - Ambient
   // 21 - GH
   // 22 - Output of outside rig
   // 23 - Output of Inside rig
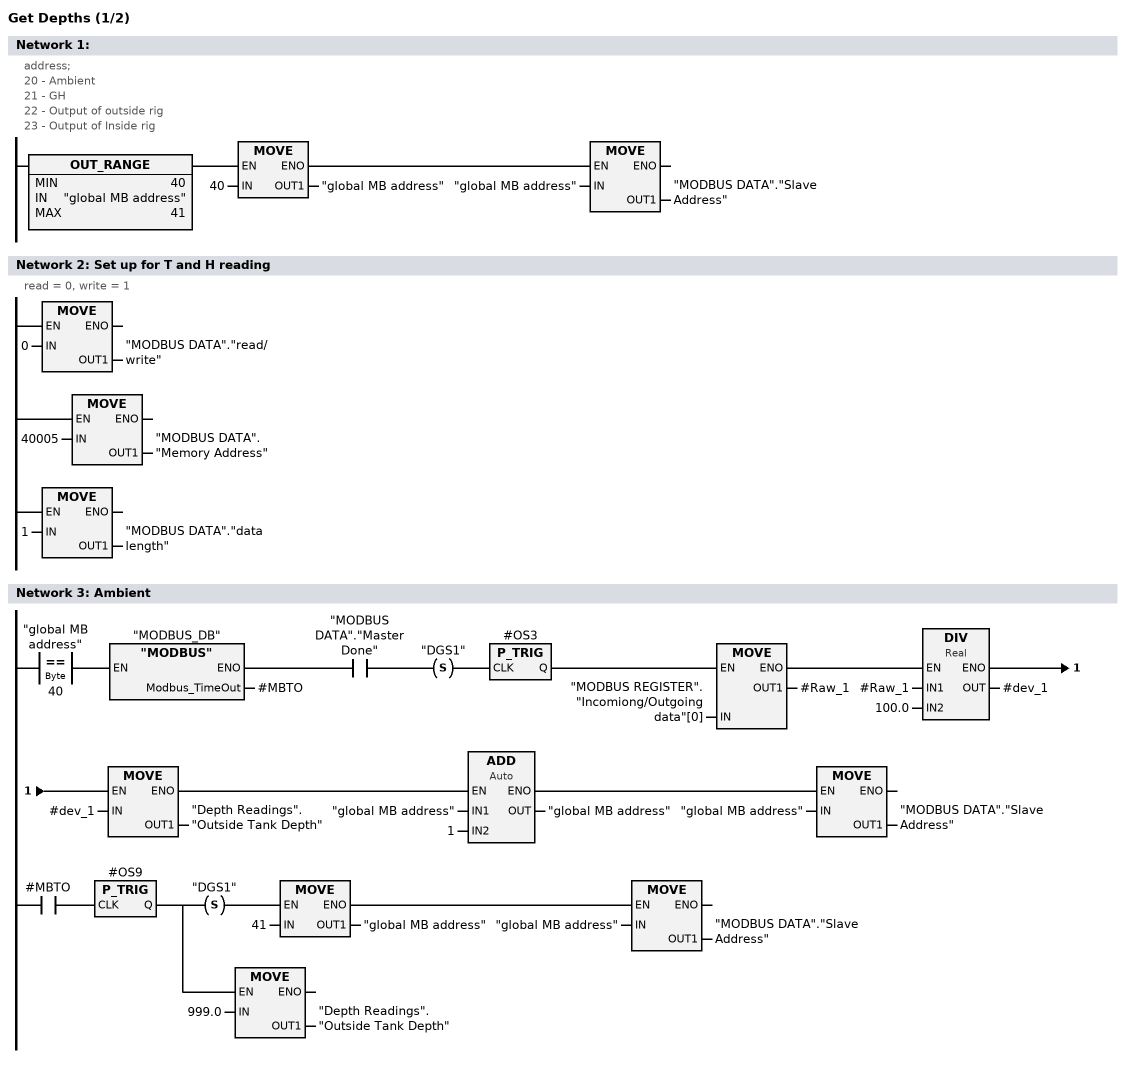
   #_w1 := ("global MB address" < 40) OR ("global MB address" > 41);
   IF #_w1 THEN
       "global MB address" := 40;
       "MODBUS DATA"."Slave Address" := "global MB address";
   END_IF;
END_REGION

REGION Network 2: Set up for T and H reading
   // read = 0, write = 1
   RUNG wire#powerrail
      Move(in := 0, out1 => "MODBUS DATA"."read/write")
   END_RUNG
   RUNG wire#powerrail
      Move(in := 40005, out1 => "MODBUS DATA"."Memory Address")
   END_RUNG
   RUNG wire#powerrail
      Move(in := 1, out1 => "MODBUS DATA"."data length")
   END_RUNG
   // the same network as SCL:
   "MODBUS DATA"."read/write" := 0;
   "MODBUS DATA"."Memory Address" := 40005;
   "MODBUS DATA"."data length" := 1;
END_REGION

REGION Network 3: Ambient
   RUNG wire#powerrail
      { S7_Templates := "SrcType := Byte" } EQ_Contact(in1 := "global MB address", in2 := 40)
      "MODBUS_DB"(Modbus_TimeOut => #MBTO)
      Contact( "MODBUS DATA"."Master Done" )
      S_Coil( "DGS1" )
      P_Trig( #OS3 )
      Move(in := "MODBUS REGISTER"."Incomiong/Outgoing data"[0], out1 => #Raw_1)
      { S7_Templates := "SrcType := Real" } Div(in1 := #Raw_1, in2 := 100.0, out => #dev_1)
      Move(in := #dev_1, out1 => "Depth Readings"."Outside Tank Depth")
      Add(in1 := "global MB address", in2 := 1, out => "global MB address")
      Move(in := "global MB address", out1 => "MODBUS DATA"."Slave Address")
   END_RUNG
   RUNG wire#powerrail
      Contact( #MBTO )
      P_Trig( #OS9 )
      wire#w1
      S_Coil( "DGS1" )
      Move(in := 41, out1 => "global MB address")
      Move(in := "global MB address", out1 => "MODBUS DATA"."Slave Address")
   END_RUNG
   RUNG wire#w1
      Move(in := 999.0, out1 => "Depth Readings"."Outside Tank Depth")
   END_RUNG
   // the same network as SCL:
   "MODBUS_DB"(EN := "global MB address" = 40, Modbus_TimeOut => #MBTO, ENO => #_w1);   // "MODBUS"
   #_w2 := #_w1 AND "MODBUS DATA"."Master Done";
   IF #_w2 THEN "DGS1" := TRUE; END_IF;
   #_w3 := #_w2 AND NOT #OS3;   // rising edge
   #OS3 := #_w2;
   IF #_w3 THEN
       #Raw_1 := "MODBUS REGISTER"."Incomiong/Outgoing data"[0];
       #dev_1 := #Raw_1 / 100.0;
       "Depth Readings"."Outside Tank Depth" := #dev_1;
       "global MB address" := "global MB address" + 1;
       "MODBUS DATA"."Slave Address" := "global MB address";
   END_IF;
   #_w4 := #MBTO AND NOT #OS9;   // rising edge
   #OS9 := #MBTO;
   IF #_w4 THEN
       "DGS1" := TRUE;
       "global MB address" := 41;
       "MODBUS DATA"."Slave Address" := "global MB address";
       "Depth Readings"."Outside Tank Depth" := 999.0;
   END_IF;
END_REGION

REGION Network 4: Greenhouse
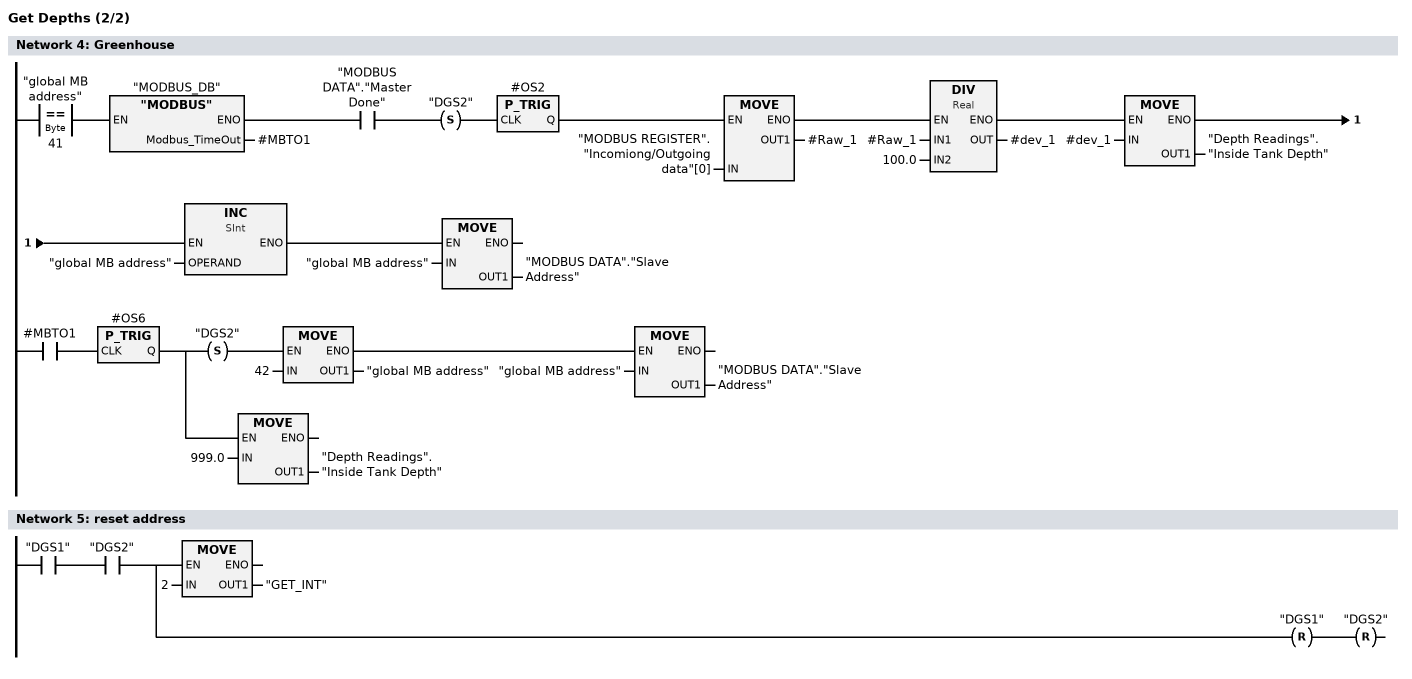
   RUNG wire#powerrail
      { S7_Templates := "SrcType := Byte" } EQ_Contact(in1 := "global MB address", in2 := 41)
      "MODBUS_DB"(Modbus_TimeOut => #MBTO1)
      Contact( "MODBUS DATA"."Master Done" )
      S_Coil( "DGS2" )
      P_Trig( #OS2 )
      Move(in := "MODBUS REGISTER"."Incomiong/Outgoing data"[0], out1 => #Raw_1)
      { S7_Templates := "SrcType := Real" } Div(in1 := #Raw_1, in2 := 100.0, out => #dev_1)
      Move(in := #dev_1, out1 => "Depth Readings"."Inside Tank Depth")
      { S7_Templates := "DestType := SInt" } Inc( "global MB address" )
      Move(in := "global MB address", out1 => "MODBUS DATA"."Slave Address")
   END_RUNG
   RUNG wire#powerrail
      Contact( #MBTO1 )
      P_Trig( #OS6 )
      wire#w1
      S_Coil( "DGS2" )
      Move(in := 42, out1 => "global MB address")
      Move(in := "global MB address", out1 => "MODBUS DATA"."Slave Address")
   END_RUNG
   RUNG wire#w1
      Move(in := 999.0, out1 => "Depth Readings"."Inside Tank Depth")
   END_RUNG
   // the same network as SCL:
   "MODBUS_DB"(EN := "global MB address" = 41, Modbus_TimeOut => #MBTO1, ENO => #_w1);   // "MODBUS"
   #_w2 := #_w1 AND "MODBUS DATA"."Master Done";
   IF #_w2 THEN "DGS2" := TRUE; END_IF;
   #_w3 := #_w2 AND NOT #OS2;   // rising edge
   #OS2 := #_w2;
   IF #_w3 THEN
       #Raw_1 := "MODBUS REGISTER"."Incomiong/Outgoing data"[0];
       #dev_1 := #Raw_1 / 100.0;
       "Depth Readings"."Inside Tank Depth" := #dev_1;
       "global MB address" := "global MB address" + 1;
       "MODBUS DATA"."Slave Address" := "global MB address";
   END_IF;
   #_w4 := #MBTO1 AND NOT #OS6;   // rising edge
   #OS6 := #MBTO1;
   IF #_w4 THEN
       "DGS2" := TRUE;
       "global MB address" := 42;
       "MODBUS DATA"."Slave Address" := "global MB address";
       "Depth Readings"."Inside Tank Depth" := 999.0;
   END_IF;
END_REGION

REGION Network 5: reset address
   RUNG wire#powerrail
      Contact( "DGS1" )
      Contact( "DGS2" )
      wire#w1
      Move(in := 2, out1 => "GET_INT")
   END_RUNG
   RUNG wire#w1
      R_Coil( "DGS1" )
      R_Coil( "DGS2" )
   END_RUNG
   // the same network as SCL:
   IF "DGS1" AND "DGS2" THEN "GET_INT" := 2; END_IF;
   #_w1 := "DGS1" AND "DGS2";
   IF #_w1 THEN
       "DGS1" := FALSE;
       "DGS2" := FALSE;
   END_IF;
END_REGION
END_FUNCTION_BLOCK

FUNCTION_BLOCK "Get Water Temp"   // FB18, LAD
{ S7_Optimized_Access := 'TRUE' }
VERSION : 0.1
   VAR
      Raw_1 : Int;
      dev_1 : Real;
      Raw_2 : Int;
      dev_2 : Real;
      MBTO : Bool;
      OS7 : Bool;
      OS6 : Bool;
      OS8 : Bool;
      OS9 : Bool;
   END_VAR
   VAR_TEMP
      OS2 : Bool;
      OS3 : Bool;
      OS4 : Bool;
      OS5 : Bool;
      MBTO1 : Bool;
      MBTO2 : Bool;
      MBTO3 : Bool;
   END_VAR
   VAR_TEMP   // added for the SCL form of the ladder/FBD networks
      _w1 : Bool;
      _w2 : Bool;
      _w3 : Bool;
      _w4 : Bool;
   END_VAR
BEGIN

REGION Network 1
   // address;
   // 20 - Ambient
   // 21 - GH
   // 22 - Output of outside rig
   // 23 - Output of Inside rig
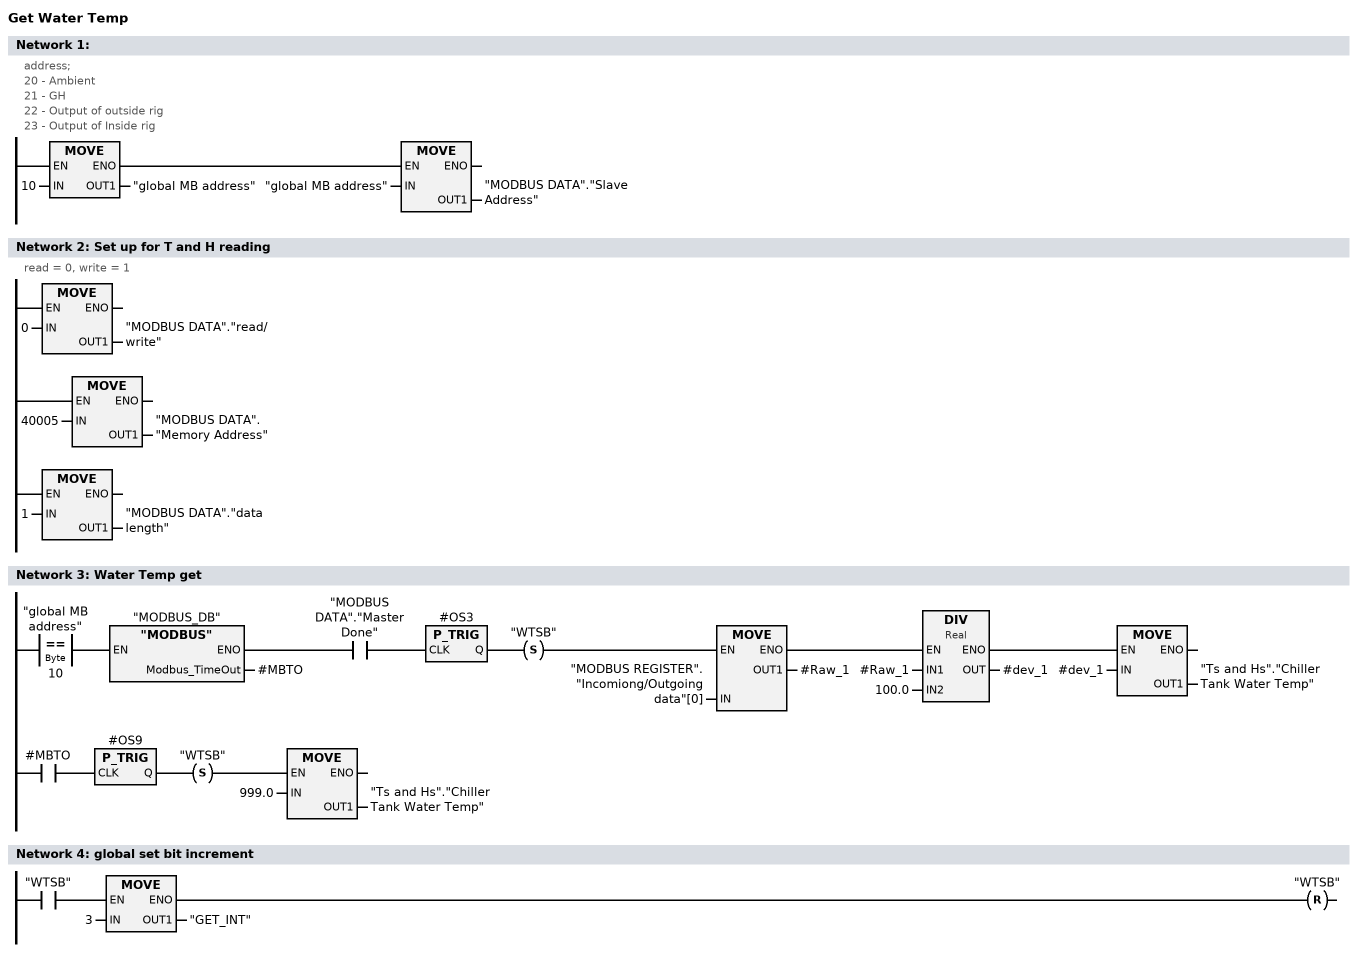
   RUNG wire#powerrail
      Move(in := 10, out1 => "global MB address")
      Move(in := "global MB address", out1 => "MODBUS DATA"."Slave Address")
   END_RUNG
   // the same network as SCL:
   "global MB address" := 10;
   "MODBUS DATA"."Slave Address" := "global MB address";
END_REGION

REGION Network 2: Set up for T and H reading
   // read = 0, write = 1
   RUNG wire#powerrail
      Move(in := 0, out1 => "MODBUS DATA"."read/write")
   END_RUNG
   RUNG wire#powerrail
      Move(in := 40005, out1 => "MODBUS DATA"."Memory Address")
   END_RUNG
   RUNG wire#powerrail
      Move(in := 1, out1 => "MODBUS DATA"."data length")
   END_RUNG
   // the same network as SCL:
   "MODBUS DATA"."read/write" := 0;
   "MODBUS DATA"."Memory Address" := 40005;
   "MODBUS DATA"."data length" := 1;
END_REGION

REGION Network 3: Water Temp get
   RUNG wire#powerrail
      { S7_Templates := "SrcType := Byte" } EQ_Contact(in1 := "global MB address", in2 := 10)
      "MODBUS_DB"(Modbus_TimeOut => #MBTO)
      Contact( "MODBUS DATA"."Master Done" )
      P_Trig( #OS3 )
      S_Coil( "WTSB" )
      Move(in := "MODBUS REGISTER"."Incomiong/Outgoing data"[0], out1 => #Raw_1)
      { S7_Templates := "SrcType := Real" } Div(in1 := #Raw_1, in2 := 100.0, out => #dev_1)
      Move(in := #dev_1, out1 => "Ts and Hs"."Chiller Tank Water Temp")
   END_RUNG
   RUNG wire#powerrail
      Contact( #MBTO )
      P_Trig( #OS9 )
      S_Coil( "WTSB" )
      Move(in := 999.0, out1 => "Ts and Hs"."Chiller Tank Water Temp")
   END_RUNG
   // the same network as SCL:
   "MODBUS_DB"(EN := "global MB address" = 10, Modbus_TimeOut => #MBTO, ENO => #_w1);   // "MODBUS"
   #_w2 := #_w1 AND "MODBUS DATA"."Master Done";
   #_w3 := #_w2 AND NOT #OS3;   // rising edge
   #OS3 := #_w2;
   IF #_w3 THEN
       "WTSB" := TRUE;
       #Raw_1 := "MODBUS REGISTER"."Incomiong/Outgoing data"[0];
       #dev_1 := #Raw_1 / 100.0;
       "Ts and Hs"."Chiller Tank Water Temp" := #dev_1;
   END_IF;
   #_w4 := #MBTO AND NOT #OS9;   // rising edge
   #OS9 := #MBTO;
   IF #_w4 THEN
       "WTSB" := TRUE;
       "Ts and Hs"."Chiller Tank Water Temp" := 999.0;
   END_IF;
END_REGION

REGION Network 4: global set bit increment
   RUNG wire#powerrail
      Contact( "WTSB" )
      Move(in := 3, out1 => "GET_INT")
      R_Coil( "WTSB" )
   END_RUNG
   // the same network as SCL:
   IF "WTSB" THEN
       "GET_INT" := 3;
       "WTSB" := FALSE;
   END_IF;
END_REGION
END_FUNCTION_BLOCK

FUNCTION_BLOCK "Update Outside Fan"   // FB19, LAD
{ S7_Optimized_Access := 'TRUE' }
VERSION : 0.1
BEGIN

REGION Network 1
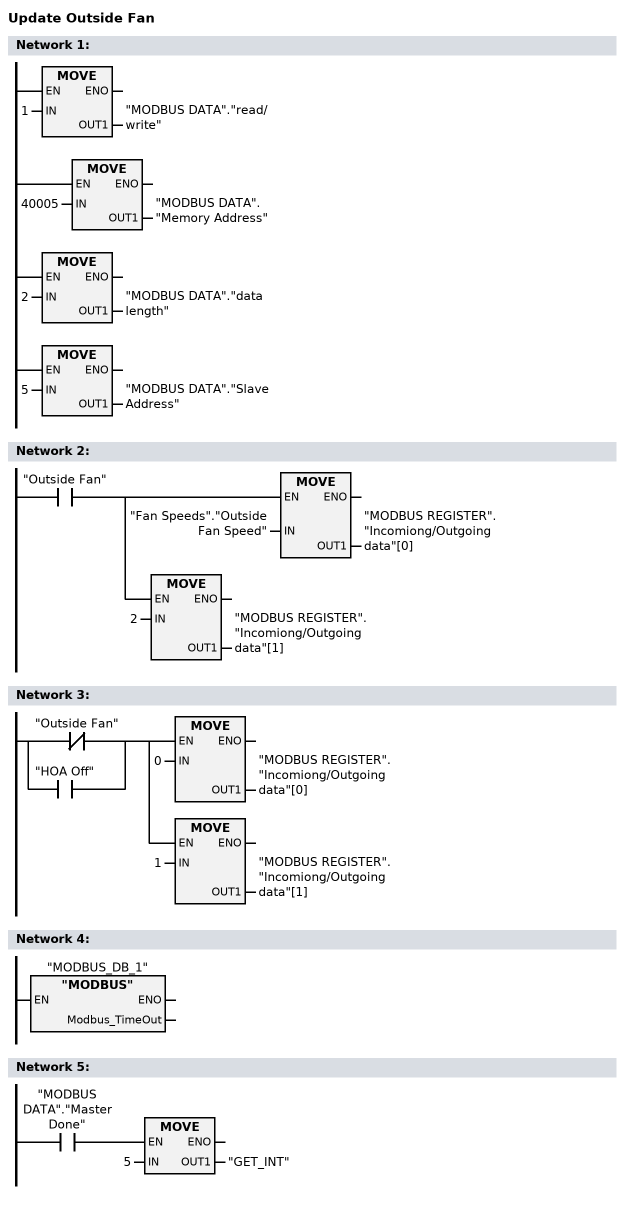
   RUNG wire#powerrail
      Move(in := 1, out1 => "MODBUS DATA"."read/write")
   END_RUNG
   RUNG wire#powerrail
      Move(in := 40005, out1 => "MODBUS DATA"."Memory Address")
   END_RUNG
   RUNG wire#powerrail
      Move(in := 2, out1 => "MODBUS DATA"."data length")
   END_RUNG
   RUNG wire#powerrail
      Move(in := 5, out1 => "MODBUS DATA"."Slave Address")
   END_RUNG
   // the same network as SCL:
   "MODBUS DATA"."read/write" := 1;
   "MODBUS DATA"."Memory Address" := 40005;
   "MODBUS DATA"."data length" := 2;
   "MODBUS DATA"."Slave Address" := 5;
END_REGION

REGION Network 2
   RUNG wire#powerrail
      Contact( "Outside Fan" )
      wire#w1
      Move(in := "Fan Speeds"."Outside Fan Speed", out1 => "MODBUS REGISTER"."Incomiong/Outgoing data"[0])
   END_RUNG
   RUNG wire#w1
      Move(in := 2, out1 => "MODBUS REGISTER"."Incomiong/Outgoing data"[1])
   END_RUNG
   // the same network as SCL:
   IF "Outside Fan" THEN
       "MODBUS REGISTER"."Incomiong/Outgoing data"[0] := "Fan Speeds"."Outside Fan Speed";
       "MODBUS REGISTER"."Incomiong/Outgoing data"[1] := 2;
   END_IF;
END_REGION

REGION Network 3
   RUNG wire#powerrail
      I_Contact( "Outside Fan" )
      wire#w1
      Move(in := 0, out1 => "MODBUS REGISTER"."Incomiong/Outgoing data"[0])
   END_RUNG
   RUNG wire#powerrail
      Contact( "HOA Off" )
   END_RUNG wire#w1
   RUNG wire#w1
      Move(in := 1, out1 => "MODBUS REGISTER"."Incomiong/Outgoing data"[1])
   END_RUNG
   // the same network as SCL:
   IF NOT "Outside Fan" OR "HOA Off" THEN
       "MODBUS REGISTER"."Incomiong/Outgoing data"[0] := 0;
       "MODBUS REGISTER"."Incomiong/Outgoing data"[1] := 1;
   END_IF;
END_REGION

REGION Network 4
   RUNG wire#powerrail
      "MODBUS_DB_1"(Modbus_TimeOut =>)
   END_RUNG
   // the same network as SCL:
   "MODBUS_DB_1"();   // "MODBUS"
END_REGION

REGION Network 5
   RUNG wire#powerrail
      Contact( "MODBUS DATA"."Master Done" )
      Move(in := 5, out1 => "GET_INT")
   END_RUNG
   // the same network as SCL:
   IF "MODBUS DATA"."Master Done" THEN "GET_INT" := 5; END_IF;
END_REGION
END_FUNCTION_BLOCK

FUNCTION_BLOCK "Update Inside Fan"   // FB20, LAD
{ S7_Optimized_Access := 'TRUE' }
VERSION : 0.1
BEGIN

REGION Network 1
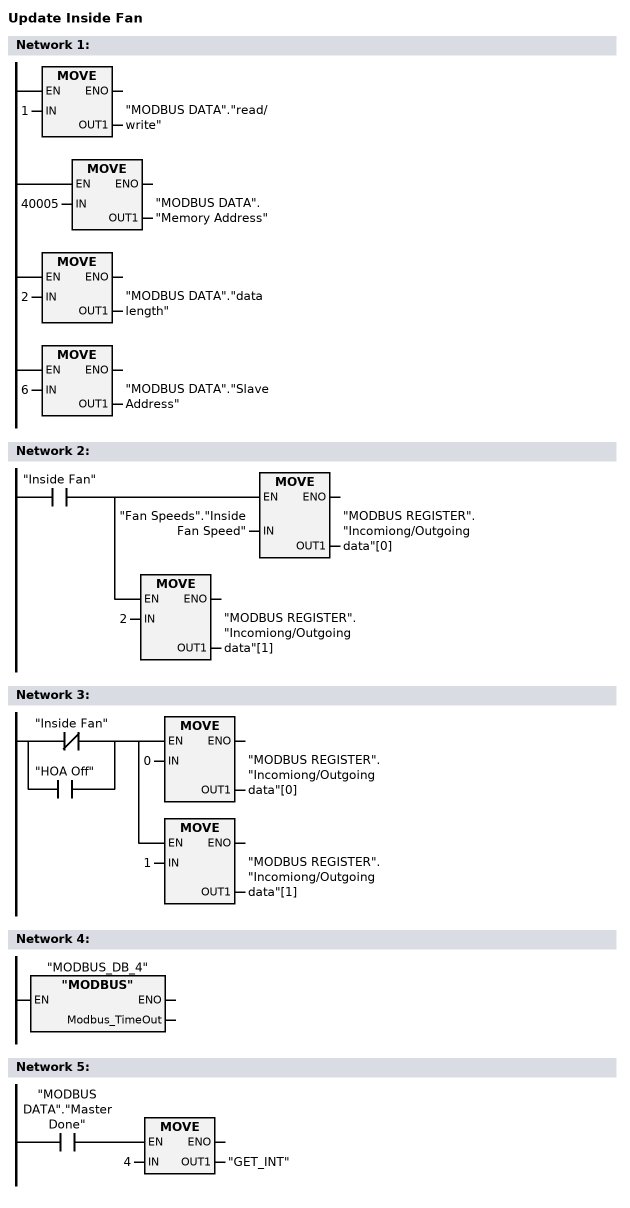
   RUNG wire#powerrail
      Move(in := 1, out1 => "MODBUS DATA"."read/write")
   END_RUNG
   RUNG wire#powerrail
      Move(in := 40005, out1 => "MODBUS DATA"."Memory Address")
   END_RUNG
   RUNG wire#powerrail
      Move(in := 2, out1 => "MODBUS DATA"."data length")
   END_RUNG
   RUNG wire#powerrail
      Move(in := 6, out1 => "MODBUS DATA"."Slave Address")
   END_RUNG
   // the same network as SCL:
   "MODBUS DATA"."read/write" := 1;
   "MODBUS DATA"."Memory Address" := 40005;
   "MODBUS DATA"."data length" := 2;
   "MODBUS DATA"."Slave Address" := 6;
END_REGION

REGION Network 2
   RUNG wire#powerrail
      Contact( "Inside Fan" )
      wire#w1
      Move(in := "Fan Speeds"."Inside Fan Speed", out1 => "MODBUS REGISTER"."Incomiong/Outgoing data"[0])
   END_RUNG
   RUNG wire#w1
      Move(in := 2, out1 => "MODBUS REGISTER"."Incomiong/Outgoing data"[1])
   END_RUNG
   // the same network as SCL:
   IF "Inside Fan" THEN
       "MODBUS REGISTER"."Incomiong/Outgoing data"[0] := "Fan Speeds"."Inside Fan Speed";
       "MODBUS REGISTER"."Incomiong/Outgoing data"[1] := 2;
   END_IF;
END_REGION

REGION Network 3
   RUNG wire#powerrail
      I_Contact( "Inside Fan" )
      wire#w1
      Move(in := 0, out1 => "MODBUS REGISTER"."Incomiong/Outgoing data"[0])
   END_RUNG
   RUNG wire#powerrail
      Contact( "HOA Off" )
   END_RUNG wire#w1
   RUNG wire#w1
      Move(in := 1, out1 => "MODBUS REGISTER"."Incomiong/Outgoing data"[1])
   END_RUNG
   // the same network as SCL:
   IF NOT "Inside Fan" OR "HOA Off" THEN
       "MODBUS REGISTER"."Incomiong/Outgoing data"[0] := 0;
       "MODBUS REGISTER"."Incomiong/Outgoing data"[1] := 1;
   END_IF;
END_REGION

REGION Network 4
   RUNG wire#powerrail
      "MODBUS_DB_4"(Modbus_TimeOut =>)
   END_RUNG
   // the same network as SCL:
   "MODBUS_DB_4"();   // "MODBUS"
END_REGION

REGION Network 5
   RUNG wire#powerrail
      Contact( "MODBUS DATA"."Master Done" )
      Move(in := 4, out1 => "GET_INT")
   END_RUNG
   // the same network as SCL:
   IF "MODBUS DATA"."Master Done" THEN "GET_INT" := 4; END_IF;
END_REGION
END_FUNCTION_BLOCK

FUNCTION_BLOCK "Outside Fan Emergancy"   // FB21, LAD
{ S7_Optimized_Access := 'TRUE' }
VERSION : 0.1
BEGIN

REGION Network 1
